gvl_p.etapa_process[0] := 'Secagem';

ELSE
	status:= 20;
END_IF

30:
IF gvl_p.arrStatusEstufas[0].prevFimSeca = systemtime_to_dt(gvl.fbGetLocalSystemTime.systemTime) THEN
	status:= 40;
	
	gvl_p.zona1setpt_019:= gvl_p.arrStatusEstufas[0].tempArm;
	gvl_p.zona2setpt_019:= gvl_p.arrStatusEstufas[0].tempArm;
	
///// GERADOR DE LOG -------------------------------------------------------------
envialog:= 'Armazenagem Iniciada ESTUFA 019';
gvl.logRegister19:= envialog;
	
gvl_p.etapa_process[0] := 'Armazenagem';

ELSE
	status:= 30;
END_IF

40:
IF gvl_p.arrStatusEstufas[0].fimArmazenagem = systemtime_to_dt(gvl.fbGetLocalSystemTime.systemTime) THEN
	status:= 50;
	
	gvl_p.arrStatusEstufas[0].start:= FALSE;
	gvl.bstartchart019:= FALSE;
	gvl.desl_aquecimento_019:= TRUE;
	fbTimeAqueci(in:=TRUE, pt:=T#1S);
	
	gvl_p.etapa_process[0] := '';
	
	gvl_p.arrStatusEstufas[0].statusInicioSecagem := '';
	gvl_p.arrStatusEstufas[0].inicioReator := '';
	gvl_p.arrStatusEstufas[0].statusFimSecagem := '';
	gvl_p.arrStatusEstufas[0].statusFimArmazenagem := '';
	gvl_p.arrStatusEstufas[0].fimSecagem:= DT#1970-1-1-0:0:0;
	gvl.endArm19:= T#0S;
	gvl.endSeca19:= T#0S;
	
	
///// GERADOR DE LOG -------------------------------------------------------------
envialog:= 'Programação Finalizada ESTUFA 019';
gvl.logRegister19:= envialog;

gvl_p.etapa_process[0]:= '';

ELSE
	status:= 40;
END_IF

45:
IF gvl_p.arrStatusEstufas[0].start THEN
status:= 50;
	
	gvl_p.arrStatusEstufas[0].start:= FALSE;
	gvl.bstartchart019:= FALSE;
	gvl.desl_aquecimento_019:= TRUE;
	fbTimeAqueci(in:=TRUE, pt:=T#1S);
	
	gvl_p.etapa_process[0] := '';
	
	gvl_p.arrStatusEstufas[0].statusInicioSecagem := '';
	gvl_p.arrStatusEstufas[0].inicioReator := '';
	gvl_p.arrStatusEstufas[0].statusFimSecagem := '';
	gvl_p.arrStatusEstufas[0].statusFimArmazenagem := '';
	gvl_p.arrStatusEstufas[0].fimSecagem:= DT#1970-1-1-0:0:0;
	gvl.endArm19:= T#0S;
	gvl.endSeca19:= T#0S;
	
///// GERADOR DE LOG -------------------------------------------------------------
envialog:= 'Programação Finalizada ESTUFA 019';
gvl.logRegister19:= envialog;

gvl_p.etapa_process[0]:= '';

ELSE
	status:= 45;
END_IF

50:
IF fbTimeAqueci.Q THEN
	status:= 0;
	
	gvl.desl_aquecimento_019:= FALSE;
	fbTimeAqueci(in:= FALSE);
	
ELSE
	status:= 50;
END_IF
END_CASE

END_PROGRAM

// ---- POUs/Rotina019_Manual.TcPOU
PROGRAM Rotina019_Manual
VAR
	status: INT;
	
	posicaoAtual: STRING;
	envialog: STRING;
	
	fbTimeVentila: ton;
	fbTimeAqueci: ton;
	
	totalManual: STRING(255);
	tempo: STRING(255);
END_VAR

fbTimeVentila();
fbTimeAqueci();

CASE status OF

0:
IF gvl_p.arrStatusEstufas[0].startManual AND STRING_TO_DT(gvl.progInicio[0]) <= systemtime_to_dt(gvl.fbGetLocalSystemTime.systemTime)  THEN
	status:= 5;
	
	gvl.bstartchart019:= TRUE;
	gvl_p.zona1setpt_019:= gvl_p.arr_CustomTime[0,1];
	gvl_p.zona2setpt_019:= gvl_p.arr_CustomTime[0,1];
	gvl.liga_ventilacao_019:= TRUE;
	fbTimeVentila(in:= TRUE, pt:=T#1S);
	
///// GERADOR DE LOG -------------------------------------------------------------

envialog:= 'Programação Manual Iniciada ESTUFA 019';
gvl.logRegister19:= envialog;

	gvl_p.etapa_process[0] := 'Inicializando';
	
ELSE
	status:= 0;
	IF gvl_p.arrStatusEstufas[0].start THEN
		gvl_p.etapa_process[0] := gvl.progInicio[0];
	END_IF
END_IF
5:
IF fbTimeVentila.Q THEN
	status:= 10;
	gvl.liga_ventilacao_019:=FALSE;
	fbTimeVentila(in:= FALSE);
ELSE
	status:= 5;
END_IF

10:
IF gvl.ventilacao_Ligada_019 THEN
	status:= 15;
	
	gvl.liga_aquecimento_019:= TRUE;
	fbTimeAqueci(in:= TRUE, pt:= T#1S);
	
///// GERADOR DE LOG -------------------------------------------------------------

envialog:= 'Aquecendo ESTUFA 019';
gvl.logRegister19:= envialog;
	
	gvl_p.etapa_process[0] := 'Aquecendo';
	
ELSE
	status:= 10;
END_IF

15:
IF fbTimeAqueci.Q THEN
	status:= 20;
	
	gvl.liga_aquecimento_019:= FALSE;
	fbTimeAqueci(in:=false);
ELSE
	status:= 15;
END_IF

20:
IF gvl.zona1atual_019 >= gvl_p.zona1setpt_019 THEN
	status:= 30;
	
gvl.progInicio[0]:= DT_TO_STRING(gvl.somaTempo);
	
///// CALCULAR FIM DA SECAGEM E DA ARMAZENAGEM --------------------------------------------------------------------------------

totalManual:= insert('T#h',INT_TO_STRING(gvl.totalManual[0]),2);
gvl_p.arrStatusEstufas[0].inicioSecagem := STRING_TO_DT(gvl.progInicio[0]);
gvl_p.arrStatusEstufas[0].fimSecagem := STRING_TO_DT(gvl.progInicio[0]) + STRING_TO_TIME(totalManual);
gvl_P.arrStatusEstufas[0].prevFimSeca := gvl_p.arrStatusEstufas[0].fimSecagem;
//gvl_p.arrStatusEstufas[0].fimArmazenagem := gvl_p.arrStatusEstufas[0].fimSecagem + gvl_p.arrStatusEstufas[0].tempoArmazenagem ;

///// IMPRIMIR A HORA E A DATA DO INICIO DA SECAGEM ---------------------------------------------------------------------------
gvl_p.arrStatusEstufas[0].statusInicioSecagem := '';
gvl_p.arrStatusEstufas[0].statusInicioSecagem := concat(gvl_p.arrStatusEstufas[0].statusInicioSecagem,gvl.hora);
gvl_p.arrStatusEstufas[0].statusInicioSecagem := concat(gvl_p.arrStatusEstufas[0].statusInicioSecagem,':');
gvl_p.arrStatusEstufas[0].statusInicioSecagem := concat(gvl_p.arrStatusEstufas[0].statusInicioSecagem,gvl.minuto);
gvl_p.arrStatusEstufas[0].statusInicioSecagem := concat(gvl_p.arrStatusEstufas[0].statusInicioSecagem,' ');
gvl_p.arrStatusEstufas[0].statusInicioSecagem := concat(gvl_p.arrStatusEstufas[0].statusInicioSecagem,gvl.dia);
gvl_p.arrStatusEstufas[0].statusInicioSecagem := concat(gvl_p.arrStatusEstufas[0].statusInicioSecagem,'/');
gvl_p.arrStatusEstufas[0].statusInicioSecagem := concat(gvl_p.arrStatusEstufas[0].statusInicioSecagem,gvl.mes);
gvl_p.arrStatusEstufas[0].statusInicioSecagem := concat(gvl_p.arrStatusEstufas[0].statusInicioSecagem,'/');
gvl_p.arrStatusEstufas[0].statusInicioSecagem := concat(gvl_p.arrStatusEstufas[0].statusInicioSecagem,gvl.ano);

//--------------------REATOR------------------------------------

IF gravarConfigPosicao_Reator.bGravarConfigPosicao_Reator THEN
	gvl_p.arrStatusEstufas[0].inicioReator := '';
	gvl_p.arrStatusEstufas[0].inicioReator := concat(gvl_p.arrStatusEstufas[0].inicioReator,gvl.hora);
	gvl_p.arrStatusEstufas[0].inicioReator := concat(gvl_p.arrStatusEstufas[0].inicioReator,':');
	gvl_p.arrStatusEstufas[0].inicioReator := concat(gvl_p.arrStatusEstufas[0].inicioReator,gvl.minuto);
	gvl_p.arrStatusEstufas[0].inicioReator := concat(gvl_p.arrStatusEstufas[0].inicioReator,' ');
	gvl_p.arrStatusEstufas[0].inicioReator := concat(gvl_p.arrStatusEstufas[0].inicioReator,gvl.dia);
	gvl_p.arrStatusEstufas[0].inicioReator := concat(gvl_p.arrStatusEstufas[0].inicioReator,'/');
	gvl_p.arrStatusEstufas[0].inicioReator := concat(gvl_p.arrStatusEstufas[0].inicioReator,gvl.mes);
	gvl_p.arrStatusEstufas[0].inicioReator := concat(gvl_p.arrStatusEstufas[0].inicioReator,'/');
	gvl_P.arrStatusEstufas[0].inicioReator := concat(gvl_p.arrStatusEstufas[0].inicioReator,gvl.ano);
END_IF

///// DECOMPOR A VARIAVEL FIM DA SECAGEM -----------------------------------------------------------------------------------------------
gvl_p.arrStatusEstufas[0].diaSec := MID(STR:= DT_TO_STRING(gvl_p.arrStatusEstufas[0].fimSecagem) , LEN:= 2, POS:=12);
gvl_p.arrStatusEstufas[0].mesSec := MID(STR:= DT_TO_STRING(gvl_p.arrStatusEstufas[0].fimSecagem), LEN:= 2, POS:=9);
gvl_p.arrStatusEstufas[0].anoSec := MID(STR:= DT_TO_STRING(gvl_p.arrStatusEstufas[0].fimSecagem), LEN:= 2, POS:=6);
gvl_p.arrStatusEstufas[0].horaSec := MID(STR:= DT_TO_STRING(gvl_p.arrStatusEstufas[0].fimSecagem), LEN:= 2, POS:=15);
gvl_p.arrStatusEstufas[0].minutoSec := MID(STR:= DT_TO_STRING(gvl_p.arrStatusEstufas[0].fimSecagem), LEN:= 2, POS:=18);

///// IMPRIMIR A HORA E A DATA DO FIM DA SECAGEM --------------------------------------------------------------------------------------------------------
gvl_p.arrStatusEstufas[0].statusFimSecagem := '';
gvl_p.arrStatusEstufas[0].statusFimSecagem := concat(gvl_p.arrStatusEstufas[0].statusFimSecagem,gvl_p.arrStatusEstufas[0].horaSec);
gvl_p.arrStatusEstufas[0].statusFimSecagem := concat(gvl_p.arrStatusEstufas[0].statusFimSecagem,':');
gvl_p.arrStatusEstufas[0].statusFimSecagem := concat(gvl_p.arrStatusEstufas[0].statusFimSecagem,gvl_p.arrStatusEstufas[0].minutoSec);
gvl_p.arrStatusEstufas[0].statusFimSecagem := concat(gvl_p.arrStatusEstufas[0].statusFimSecagem,' ');
gvl_p.arrStatusEstufas[0].statusFimSecagem := concat(gvl_p.arrStatusEstufas[0].statusFimSecagem,gvl_p.arrStatusEstufas[0].diaSec);
gvl_p.arrStatusEstufas[0].statusFimSecagem := concat(gvl_p.arrStatusEstufas[0].statusFimSecagem,'/');
gvl_p.arrStatusEstufas[0].statusFimSecagem := concat(gvl_p.arrStatusEstufas[0].statusFimSecagem,gvl_p.arrStatusEstufas[0].mesSec);
gvl_p.arrStatusEstufas[0].statusFimSecagem := concat(gvl_p.arrStatusEstufas[0].statusFimSecagem,'/');
gvl_p.arrStatusEstufas[0].statusFimSecagem := concat(gvl_p.arrStatusEstufas[0].statusFimSecagem,gvl_p.arrStatusEstufas[0].anoSec);


///// GERADOR DE LOG -------------------------------------------------------------
envialog:= 'Inicio T1 ESTUFA 019';
gvl.logRegister19:= envialog;

gvl_p.etapa_process[0]:= 'T1';

ELSE
	IF gvl_p.arr_CustomTime[1,1] = 0 THEN
		status:= 45;
	END_IF
	status:= 20;
END_IF

30:
tempo:= insert('T#h',INT_TO_STRING(gvl_p.arr_CustomTime[1,1]),2);
IF STRING_TO_DT(gvl.progInicio[0]) + STRING_TO_TIME(tempo) = systemtime_to_dt(gvl.fbGetLocalSystemTime.systemTime) THEN
	status:= 31;
	
	gvl_p.zona1setpt_019:= gvl_p.arr_CustomTime[0,2];
	gvl_p.zona2setpt_019:= gvl_p.arr_CustomTime[0,2];
	gvl.progInicio[0]:= DT_TO_STRING(STRING_TO_DT(gvl.progInicio[0]) + STRING_TO_TIME(tempo));
	
///// GERADOR DE LOG -------------------------------------------------------------
envialog:= 'Inicio T2 ESTUFA 019';
gvl.logRegister19:= envialog;

gvl_p.etapa_process[0]:= 'T2';
	
ELSE
	status:= 30;
END_IF

31:
tempo:= insert('T#h',INT_TO_STRING(gvl_p.arr_CustomTime[1,2]),2);
IF STRING_TO_DT(gvl.progInicio[0]) + STRING_TO_TIME(tempo) = systemtime_to_dt(gvl.fbGetLocalSystemTime.systemTime) THEN
	status:= 32;
	
	gvl_p.zona1setpt_019:= gvl_p.arr_CustomTime[0,3];
	gvl_p.zona2setpt_019:= gvl_p.arr_CustomTime[0,3];
	gvl.progInicio[0]:= DT_TO_STRING(STRING_TO_DT(gvl.progInicio[0]) + STRING_TO_TIME(tempo));
	
///// GERADOR DE LOG -------------------------------------------------------------
envialog:= 'Inicio T3 ESTUFA 019';
gvl.logRegister19:= envialog;

gvl_p.etapa_process[0]:= 'T3';
	
ELSE
	IF gvl_p.arr_CustomTime[1,2] = 0 THEN
		status:= 45;
	END_IF
	status:= 31;
END_IF

32:
tempo:= insert('T#h',INT_TO_STRING(gvl_p.arr_CustomTime[1,3]),2);
IF STRING_TO_DT(gvl.progInicio[0]) + STRING_TO_TIME(tempo) = systemtime_to_dt(gvl.fbGetLocalSystemTime.systemTime) THEN
	status:= 33;
	
	gvl_p.zona1setpt_019:= gvl_p.arr_CustomTime[0,4];
	gvl_p.zona2setpt_019:= gvl_p.arr_CustomTime[0,4];
	gvl.progInicio[0]:= DT_TO_STRING(STRING_TO_DT(gvl.progInicio[0]) + STRING_TO_TIME(tempo));
	
///// GERADOR DE LOG -------------------------------------------------------------
envialog:= 'Inicio T4 ESTUFA 019';
gvl.logRegister19:= envialog;

gvl_p.etapa_process[0]:= 'T4';
	
ELSE
	IF gvl_p.arr_CustomTime[1,3] = 0 THEN
		status:= 45;
	END_IF
	status:= 32;
END_IF

33:
tempo:= insert('T#h',INT_TO_STRING(gvl_p.arr_CustomTime[1,4]),2);
IF STRING_TO_DT(gvl.progInicio[0]) + STRING_TO_TIME(tempo) = systemtime_to_dt(gvl.fbGetLocalSystemTime.systemTime) THEN
	status:= 34;
	
	gvl_p.zona1setpt_019:= gvl_p.arr_CustomTime[0,5];
	gvl_p.zona2setpt_019:= gvl_p.arr_CustomTime[0,5];
	gvl.progInicio[0]:= DT_TO_STRING(STRING_TO_DT(gvl.progInicio[0]) + STRING_TO_TIME(tempo));
	
///// GERADOR DE LOG -------------------------------------------------------------
envialog:= 'Inicio T5 ESTUFA 019';
gvl.logRegister19:= envialog;

gvl_p.etapa_process[0]:= 'T5';
	
ELSE
	IF gvl_p.arr_CustomTime[1,4] = 0 THEN
		status:= 45;
	END_IF
	status:= 33;
END_IF

34:
tempo:= insert('T#h',INT_TO_STRING(gvl_p.arr_CustomTime[1,5]),2);
IF STRING_TO_DT(gvl.progInicio[0]) + STRING_TO_TIME(tempo) = systemtime_to_dt(gvl.fbGetLocalSystemTime.systemTime) THEN
	status:= 35;
	
	gvl_p.zona1setpt_019:= gvl_p.arr_CustomTime[0,6];
	gvl_p.zona2setpt_019:= gvl_p.arr_CustomTime[0,6];
	gvl.progInicio[0]:= DT_TO_STRING(STRING_TO_DT(gvl.progInicio[0]) + STRING_TO_TIME(tempo));
	
///// GERADOR DE LOG -------------------------------------------------------------
envialog:= 'Inicio T6 ESTUFA 019';
gvl.logRegister19:= envialog;

gvl_p.etapa_process[0]:= 'T6';
	
ELSE
	IF gvl_p.arr_CustomTime[1,5] = 0 THEN
		status:= 45;
	END_IF
	status:= 34;
END_IF

35:
tempo:= insert('T#h',INT_TO_STRING(gvl_p.arr_CustomTime[1,6]),2);
IF STRING_TO_DT(gvl.progInicio[0]) + STRING_TO_TIME(tempo) = systemtime_to_dt(gvl.fbGetLocalSystemTime.systemTime) THEN
	status:= 36;
	
	gvl_p.zona1setpt_019:= gvl_p.arr_CustomTime[0,7];
	gvl_p.zona2setpt_019:= gvl_p.arr_CustomTime[0,7];
	gvl.progInicio[0]:= DT_TO_STRING(STRING_TO_DT(gvl.progInicio[0]) + STRING_TO_TIME(tempo));
	
///// GERADOR DE LOG -------------------------------------------------------------
envialog:= 'Inicio T7 ESTUFA 019';
gvl.logRegister19:= envialog;

gvl_p.etapa_process[0]:= 'T7';
	
ELSE
	IF gvl_p.arr_CustomTime[1,6] = 0 THEN
		status:= 45;
	END_IF
	status:= 35;
END_IF

36:
tempo:= insert('T#h',INT_TO_STRING(gvl_p.arr_CustomTime[1,7]),2);
IF STRING_TO_DT(gvl.progInicio[0]) + STRING_TO_TIME(tempo) = systemtime_to_dt(gvl.fbGetLocalSystemTime.systemTime) THEN
	status:= 37;
	
	gvl_p.zona1setpt_019:= gvl_p.arr_CustomTime[0,8];
	gvl_p.zona2setpt_019:= gvl_p.arr_CustomTime[0,8];
	gvl.progInicio[0]:= DT_TO_STRING(STRING_TO_DT(gvl.progInicio[0]) + STRING_TO_TIME(tempo));
	
///// GERADOR DE LOG -------------------------------------------------------------
envialog:= 'Inicio T8 ESTUFA 019';
gvl.logRegister19:= envialog;

gvl_p.etapa_process[0]:= 'T8';
	
ELSE
	IF gvl_p.arr_CustomTime[1,7] = 0 THEN
		status:= 45;
	END_IF
	status:= 36;
END_IF

37:
tempo:= insert('T#h',INT_TO_STRING(gvl_p.arr_CustomTime[1,8]),2);
IF STRING_TO_DT(gvl.progInicio[0]) + STRING_TO_TIME(tempo) = systemtime_to_dt(gvl.fbGetLocalSystemTime.systemTime) THEN
	status:= 38;
	
	gvl_p.zona1setpt_019:= gvl_p.arr_CustomTime[0,9];
	gvl_p.zona2setpt_019:= gvl_p.arr_CustomTime[0,9];
	gvl.progInicio[0]:= DT_TO_STRING(STRING_TO_DT(gvl.progInicio[0]) + STRING_TO_TIME(tempo));
	
///// GERADOR DE LOG -------------------------------------------------------------
envialog:= 'Inicio T9 ESTUFA 019';
gvl.logRegister19:= envialog;

gvl_p.etapa_process[0]:= 'T9';
	
ELSE
	IF gvl_p.arr_CustomTime[1,8] = 0 THEN
		status:= 45;
	END_IF
	status:= 37;
END_IF

38:
tempo:= insert('T#h',INT_TO_STRING(gvl_p.arr_CustomTime[1,9]),2);
IF STRING_TO_DT(gvl.progInicio[0]) + STRING_TO_TIME(tempo) = systemtime_to_dt(gvl.fbGetLocalSystemTime.systemTime) THEN
	status:= 40;
	
	gvl_p.zona1setpt_019:= gvl_p.arr_CustomTime[0,10];
	gvl_p.zona2setpt_019:= gvl_p.arr_CustomTime[0,10];
	gvl.progInicio[0]:= DT_TO_STRING(STRING_TO_DT(gvl.progInicio[0]) + STRING_TO_TIME(tempo));
	
///// GERADOR DE LOG -------------------------------------------------------------
envialog:= 'Inicio T10 ESTUFA 019';
gvl.logRegister19:= envialog;

gvl_p.etapa_process[0]:= 'T10';
	
ELSE
	IF gvl_p.arr_CustomTime[1,9] = 0 THEN
		status:= 45;
	END_IF
	status:= 38;
END_IF

40:
tempo:= insert('T#h',INT_TO_STRING(gvl_p.arr_CustomTime[1,10]),2);
IF STRING_TO_DT(gvl.progInicio[0]) + STRING_TO_TIME(tempo) = systemtime_to_dt(gvl.fbGetLocalSystemTime.systemTime) THEN
	status:= 50;
	
	gvl_p.arrStatusEstufas[0].startManual:= FALSE;
	gvl.bstartchart019:= FALSE;
	gvl.desl_aquecimento_019:= TRUE;
	fbTimeAqueci(in:=TRUE, pt:=T#1S);
	
	gvl_p.etapa_process[0] := '';
	
	gvl_p.arrStatusEstufas[0].statusInicioSecagem := '';
	gvl_p.arrStatusEstufas[0].inicioReator := '';
	gvl_p.arrStatusEstufas[0].statusFimSecagem := '';
	gvl_p.arrStatusEstufas[0].statusFimArmazenagem := '';
	gvl_p.arrStatusEstufas[0].fimSecagem:= DT#1970-1-1-0:0:0;
	gvl.endArm19:= T#0S;
	gvl.endSeca19:= T#0S;
	
///// GERADOR DE LOG -------------------------------------------------------------
envialog:= 'Programação Finalizada ESTUFA 019';
gvl.logRegister19:= envialog;

gvl_p.etapa_process[0]:= '';

ELSE
	IF gvl_p.arr_CustomTime[1,10] = 0 THEN
		status:= 45;
	END_IF
	status:= 40;
END_IF

45:
IF gvl_p.arrStatusEstufas[0].startManual THEN
status:= 50;
	
	gvl_p.arrStatusEstufas[0].startManual:= FALSE;
	gvl.bstartchart019:= FALSE;
	gvl.desl_aquecimento_019:= TRUE;
	fbTimeAqueci(in:=TRUE, pt:=T#1S);
	
	gvl_p.etapa_process[0] := '';
	
	gvl_p.arrStatusEstufas[0].statusInicioSecagem := '';
	gvl_p.arrStatusEstufas[0].inicioReator := '';
	gvl_p.arrStatusEstufas[0].statusFimSecagem := '';
	gvl_p.arrStatusEstufas[0].statusFimArmazenagem := '';
	gvl_p.arrStatusEstufas[0].fimSecagem:= DT#1970-1-1-0:0:0;
	gvl.endArm19:= T#0S;
	gvl.endSeca19:= T#0S;
	
///// GERADOR DE LOG -------------------------------------------------------------
envialog:= 'Programação Finalizada ESTUFA 019';
gvl.logRegister19:= envialog;

gvl_p.etapa_process[0]:= '';

ELSE
	status:= 45;
END_IF

50:
IF fbTimeAqueci.Q THEN
	status:= 0;
	
	gvl.desl_aquecimento_019:= FALSE;
	fbTimeAqueci(in:= FALSE);
	
ELSE
	status:= 50;
END_IF
END_CASE

END_PROGRAM

// ---- POUs/Rotina020.TcPOU
PROGRAM Rotina020
VAR
	status: INT;
	
	posicaoAtual: STRING;
	envialog: STRING;
	
	fbTimeVentila: ton;
	fbTimeAqueci: ton;
	
	a: INT;
END_VAR

fbTimeVentila();
fbTimeAqueci();
a:=1;

CASE status OF

0:
IF gvl_p.arrStatusEstufas[a].start AND STRING_TO_DT(gvl.progInicio[a]) <= systemtime_to_dt(gvl.fbGetLocalSystemTime.systemTime)  THEN
	status:= 5;
	
	gvl.bstartchart020:= TRUE;
	gvl_p.zona1setpt_020:= gvl_p.arrStatusEstufas[a].tempSeca;
	gvl_p.zona2setpt_020:= gvl_p.arrStatusEstufas[a].tempSeca;
	gvl.liga_ventilacao_020:= TRUE;
	fbTimeVentila(in:= TRUE, pt:=T#1S);

///// GERADOR DE LOG -------------------------------------------------------------

envialog:= 'Inicializando Programação ESTUFA 020';
gvl.logRegister20:= envialog;
	
	gvl_p.etapa_process[a] := 'Inicializando';
	
ELSE
	status:= 0;
	IF gvl_p.arrStatusEstufas[a].start THEN
		gvl_p.etapa_process[a] := gvl.progInicio[a];
	END_IF
END_IF

5:
IF fbTimeVentila.Q THEN
	status:= 10;
	gvl.liga_ventilacao_020:=FALSE;
	fbTimeVentila(in:= FALSE);
ELSE
	status:= 5;
END_IF

10:
IF gvl.ventilacao_Ligada_020 THEN
	status:= 15;
	
	gvl.liga_aquecimento_020:= TRUE;
	fbTimeAqueci(in:= TRUE, pt:= T#1S);
	
///// GERADOR DE LOG -------------------------------------------------------------

envialog:= 'Aquecendo ESTUFA 020';
gvl.logRegister20:= envialog;

	gvl_p.etapa_process[a] := 'Aquecendo';
	
ELSE
	status:= 10;
END_IF

15:
IF fbTimeAqueci.Q THEN
	status:= 20;
	
	gvl.liga_aquecimento_020:= FALSE;
	fbTimeAqueci(in:=false);
ELSE
	status:= 15;
END_IF

20:
IF gvl.zona1atual_020 >= gvl_p.zona1setpt_020 THEN
	status:= 30;

gvl.progInicio[a]:= DT_TO_STRING(gvl.somaTempo);
	
///// CALCULAR FIM DA SECAGEM E DA ARMAZENAGEM --------------------------------------------------------------------------------
gvl_p.arrStatusEstufas[a].inicioSecagem := STRING_TO_DT(gvl.progInicio[a]);
gvl_p.arrStatusEstufas[a].fimSecagem := STRING_TO_DT(gvl.progInicio[a]) + gvl_p.arrStatusEstufas[a].tempoSecagem;
gvl_P.arrStatusEstufas[a].prevFimSeca := gvl_p.arrStatusEstufas[a].fimSecagem;
gvl_p.arrStatusEstufas[a].fimArmazenagem := gvl_p.arrStatusEstufas[a].fimSecagem + gvl_p.arrStatusEstufas[a].tempoArmazenagem ;

///// IMPRIMIR A HORA E A DATA DO INICIO DA SECAGEM ---------------------------------------------------------------------------
gvl_p.arrStatusEstufas[a].statusInicioSecagem := '';
gvl_p.arrStatusEstufas[a].statusInicioSecagem := concat(gvl_p.arrStatusEstufas[a].statusInicioSecagem,gvl.hora);
gvl_p.arrStatusEstufas[a].statusInicioSecagem := concat(gvl_p.arrStatusEstufas[a].statusInicioSecagem,':');
gvl_p.arrStatusEstufas[a].statusInicioSecagem := concat(gvl_p.arrStatusEstufas[a].statusInicioSecagem,gvl.minuto);
gvl_p.arrStatusEstufas[a].statusInicioSecagem := concat(gvl_p.arrStatusEstufas[a].statusInicioSecagem,' ');
gvl_p.arrStatusEstufas[a].statusInicioSecagem := concat(gvl_p.arrStatusEstufas[a].statusInicioSecagem,gvl.dia);
gvl_p.arrStatusEstufas[a].statusInicioSecagem := concat(gvl_p.arrStatusEstufas[a].statusInicioSecagem,'/');
gvl_p.arrStatusEstufas[a].statusInicioSecagem := concat(gvl_p.arrStatusEstufas[a].statusInicioSecagem,gvl.mes);
gvl_p.arrStatusEstufas[a].statusInicioSecagem := concat(gvl_p.arrStatusEstufas[a].statusInicioSecagem,'/');
gvl_p.arrStatusEstufas[a].statusInicioSecagem := concat(gvl_p.arrStatusEstufas[a].statusInicioSecagem,gvl.ano);

//--------------------REATOR------------------------------------

IF gravarConfigPosicao_Reator.bGravarConfigPosicao_Reator THEN
	gvl_p.arrStatusEstufas[a].inicioReator := '';
	gvl_p.arrStatusEstufas[a].inicioReator := concat(gvl_p.arrStatusEstufas[a].inicioReator,gvl.hora);
	gvl_p.arrStatusEstufas[a].inicioReator := concat(gvl_p.arrStatusEstufas[a].inicioReator,':');
	gvl_p.arrStatusEstufas[a].inicioReator := concat(gvl_p.arrStatusEstufas[a].inicioReator,gvl.minuto);
	gvl_p.arrStatusEstufas[a].inicioReator := concat(gvl_p.arrStatusEstufas[a].inicioReator,' ');
	gvl_p.arrStatusEstufas[a].inicioReator := concat(gvl_p.arrStatusEstufas[a].inicioReator,gvl.dia);
	gvl_p.arrStatusEstufas[a].inicioReator := concat(gvl_p.arrStatusEstufas[a].inicioReator,'/');
	gvl_p.arrStatusEstufas[a].inicioReator := concat(gvl_p.arrStatusEstufas[a].inicioReator,gvl.mes);
	gvl_p.arrStatusEstufas[a].inicioReator := concat(gvl_p.arrStatusEstufas[a].inicioReator,'/');
	gvl_P.arrStatusEstufas[a].inicioReator := concat(gvl_p.arrStatusEstufas[a].inicioReator,gvl.ano);
END_IF

///// DECOMPOR A VARIAVEL FIM DA SECAGEM -----------------------------------------------------------------------------------------------
gvl_p.arrStatusEstufas[a].diaSec := MID(STR:= DT_TO_STRING(gvl_p.arrStatusEstufas[a].fimSecagem) , LEN:= 2, POS:=12);
gvl_p.arrStatusEstufas[a].mesSec := MID(STR:= DT_TO_STRING(gvl_p.arrStatusEstufas[a].fimSecagem), LEN:= 2, POS:=9);
gvl_p.arrStatusEstufas[a].anoSec := MID(STR:= DT_TO_STRING(gvl_p.arrStatusEstufas[a].fimSecagem), LEN:= 2, POS:=6);
gvl_p.arrStatusEstufas[a].horaSec := MID(STR:= DT_TO_STRING(gvl_p.arrStatusEstufas[a].fimSecagem), LEN:= 2, POS:=15);
gvl_p.arrStatusEstufas[a].minutoSec := MID(STR:= DT_TO_STRING(gvl_p.arrStatusEstufas[a].fimSecagem), LEN:= 2, POS:=18);

///// IMPRIMIR A HORA E A DATA DO FIM DA SECAGEM --------------------------------------------------------------------------------------------------------
gvl_p.arrStatusEstufas[a].statusFimSecagem := '';
gvl_p.arrStatusEstufas[a].statusFimSecagem := concat(gvl_p.arrStatusEstufas[a].statusFimSecagem,gvl_p.arrStatusEstufas[a].horaSec);
gvl_p.arrStatusEstufas[a].statusFimSecagem := concat(gvl_p.arrStatusEstufas[a].statusFimSecagem,':');
gvl_p.arrStatusEstufas[a].statusFimSecagem := concat(gvl_p.arrStatusEstufas[a].statusFimSecagem,gvl_p.arrStatusEstufas[a].minutoSec);
gvl_p.arrStatusEstufas[a].statusFimSecagem := concat(gvl_p.arrStatusEstufas[a].statusFimSecagem,' ');
gvl_p.arrStatusEstufas[a].statusFimSecagem := concat(gvl_p.arrStatusEstufas[a].statusFimSecagem,gvl_p.arrStatusEstufas[a].diaSec);
gvl_p.arrStatusEstufas[a].statusFimSecagem := concat(gvl_p.arrStatusEstufas[a].statusFimSecagem,'/');
gvl_p.arrStatusEstufas[a].statusFimSecagem := concat(gvl_p.arrStatusEstufas[a].statusFimSecagem,gvl_p.arrStatusEstufas[a].mesSec);
gvl_p.arrStatusEstufas[a].statusFimSecagem := concat(gvl_p.arrStatusEstufas[a].statusFimSecagem,'/');
gvl_p.arrStatusEstufas[a].statusFimSecagem := concat(gvl_p.arrStatusEstufas[a].statusFimSecagem,gvl_p.arrStatusEstufas[a].anoSec);

///// DECOMPOR A VARIAVEL FIM DA ARMAZENAGEM -------------------------------------------------------------------------------------------
gvl_p.arrStatusEstufas[a].diaArm := MID(STR:= DT_TO_STRING(gvl_p.arrStatusEstufas[a].fimArmazenagem) , LEN:= 2, POS:=12);
gvl_p.arrStatusEstufas[a].mesArm := MID(STR:= DT_TO_STRING(gvl_p.arrStatusEstufas[a].fimArmazenagem), LEN:= 2, POS:=9);
gvl_p.arrStatusEstufas[a].anoArm := MID(STR:= DT_TO_STRING(gvl_P.arrStatusEstufas[a].fimArmazenagem), LEN:= 2, POS:=6);
gvl_p.arrStatusEstufas[a].horaArm := MID(STR:= DT_TO_STRING(gvl_P.arrStatusEstufas[a].fimArmazenagem), LEN:= 2, POS:=15);
gvl_p.arrStatusEstufas[a].minutoArm := MID(STR:= DT_TO_STRING(gvl_p.arrStatusEstufas[a].fimArmazenagem), LEN:= 2, POS:=18);

///// IMPRIMIR A HORA E A DATA DO FIM DA ARMAZENAGEM -----------------------------------------------------------------------------------------------------------
gvl_p.arrStatusEstufas[a].statusFimArmazenagem := '';
gvl_p.arrStatusEstufas[a].statusFimArmazenagem := concat(gvl_p.arrStatusEstufas[a].statusFimArmazenagem,gvl_p.arrStatusEstufas[a].horaArm);
gvl_p.arrStatusEstufas[a].statusFimArmazenagem := concat(gvl_p.arrStatusEstufas[a].statusFimArmazenagem,':');
gvl_p.arrStatusEstufas[a].statusFimArmazenagem := concat(gvl_p.arrStatusEstufas[a].statusFimArmazenagem,gvl_p.arrStatusEstufas[a].minutoArm);
gvl_p.arrStatusEstufas[a].statusFimArmazenagem := concat(gvl_p.arrStatusEstufas[a].statusFimArmazenagem,' ');
gvl_p.arrStatusEstufas[a].statusFimArmazenagem := concat(gvl_p.arrStatusEstufas[a].statusFimArmazenagem,gvl_p.arrStatusEstufas[a].diaArm);
gvl_p.arrStatusEstufas[a].statusFimArmazenagem := concat(gvl_p.arrStatusEstufas[a].statusFimArmazenagem,'/');
gvl_p.arrStatusEstufas[a].statusFimArmazenagem := concat(gvl_p.arrStatusEstufas[a].statusFimArmazenagem,gvl_p.arrStatusEstufas[a].mesArm);
gvl_p.arrStatusEstufas[a].statusFimArmazenagem := concat(gvl_p.arrStatusEstufas[a].statusFimArmazenagem,'/');
gvl_p.arrStatusEstufas[a].statusFimArmazenagem := concat(gvl_p.arrStatusEstufas[a].statusFimArmazenagem,gvl_p.arrStatusEstufas[a].anoArm);

///// GERADOR DE LOG -------------------------------------------------------------
envialog:= 'Secagem Iniciada ESTUFA 020';
gvl.logRegister20:= envialog;

gvl_p.etapa_process[a] := 'Secagem';

ELSE
	status:= 20;
END_IF

30:
IF gvl_p.arrStatusEstufas[a].prevFimSeca = systemtime_to_dt(gvl.fbGetLocalSystemTime.systemTime) THEN
	status:= 40;
	
	gvl_p.zona1setpt_020:= gvl_p.arrStatusEstufas[a].tempArm;
	gvl_p.zona2setpt_020:= gvl_p.arrStatusEstufas[a].tempArm;
	
///// GERADOR DE LOG -------------------------------------------------------------
envialog:= 'Armazenagem Iniciada ESTUFA 020';
gvl.logRegister20:= envialog;
	
gvl_p.etapa_process[a] := 'Armazenagem';

ELSE
	status:= 30;
END_IF

40:
IF gvl_p.arrStatusEstufas[a].fimArmazenagem = systemtime_to_dt(gvl.fbGetLocalSystemTime.systemTime) THEN
	status:= 50;
	
	gvl_p.arrStatusEstufas[a].start:= FALSE;
	gvl.bstartchart020:= FALSE;
	gvl.desl_aquecimento_020:= TRUE;
	fbTimeAqueci(in:=TRUE, pt:=T#1S);
	
	gvl_p.etapa_process[a] := '';
	
	gvl_p.arrStatusEstufas[a].statusInicioSecagem := '';
	gvl_p.arrStatusEstufas[a].inicioReator := '';
	gvl_p.arrStatusEstufas[a].statusFimSecagem := '';
	gvl_p.arrStatusEstufas[a].statusFimArmazenagem := '';
	gvl_p.arrStatusEstufas[a].fimSecagem:= DT#1970-1-1-0:0:0;
	gvl.endArm20:= T#0S;
	gvl.endSeca20:= T#0S;
	
	
///// GERADOR DE LOG -------------------------------------------------------------
envialog:= 'Programação Finalizada ESTUFA 020';
gvl.logRegister20:= envialog;

gvl_p.etapa_process[1]:= '';

ELSE
	status:= 40;
END_IF

45:
IF gvl_p.arrStatusEstufas[a].start THEN
status:= 50;
	
	gvl_p.arrStatusEstufas[a].start:= FALSE;
	gvl.bstartchart020:= FALSE;
	gvl.desl_aquecimento_020:= TRUE;
	fbTimeAqueci(in:=TRUE, pt:=T#1S);
	
	gvl_p.etapa_process[a] := '';
	
	gvl_p.arrStatusEstufas[a].statusInicioSecagem := '';
	gvl_p.arrStatusEstufas[a].inicioReator := '';
	gvl_p.arrStatusEstufas[a].statusFimSecagem := '';
	gvl_p.arrStatusEstufas[a].statusFimArmazenagem := '';
	gvl_p.arrStatusEstufas[a].fimSecagem:= DT#1970-1-1-0:0:0;
	gvl.endArm20:= T#0S;
	gvl.endSeca20:= T#0S;
	
///// GERADOR DE LOG -------------------------------------------------------------
envialog:= 'Programação Finalizada ESTUFA 020';
gvl.logRegister20:= envialog;

gvl_p.etapa_process[1]:= '';

ELSE
	status:= 45;
END_IF

50:
IF fbTimeAqueci.Q THEN
	status:= 0;
	
	gvl.desl_aquecimento_020:= FALSE;
	fbTimeAqueci(in:= FALSE);
	
ELSE
	status:= 50;
END_IF
END_CASE

END_PROGRAM

// ---- POUs/Rotina020_Manual.TcPOU
PROGRAM Rotina020_Manual
VAR
	status: INT;
	
	posicaoAtual: STRING;
	envialog: STRING;
	
	fbTimeVentila: ton;
	fbTimeAqueci: ton;
	
	totalManual: STRING(255);
	tempo: STRING(255);
	
	Estufa: INT;
	
END_VAR

fbTimeVentila();
fbTimeAqueci();
Estufa:= 1;

CASE status OF

0:
IF gvl_p.arrStatusEstufas[Estufa].startManual AND STRING_TO_DT(gvl.progInicio[Estufa]) <= systemtime_to_dt(gvl.fbGetLocalSystemTime.systemTime)  THEN
	status:= 5;
	
	gvl.bstartchart020:= TRUE;
	gvl_p.zona1setpt_020:= gvl_p.arr_CustomTime_020[0,1];
	gvl_p.zona2setpt_020:= gvl_p.arr_CustomTime_020[0,1];
	gvl.liga_ventilacao_020:= TRUE;
	fbTimeVentila(in:= TRUE, pt:=T#1S);
	
///// GERADOR DE LOG -------------------------------------------------------------

envialog:= 'Programação Manual Iniciada ESTUFA 020';
gvl.logRegister20:= envialog;

	gvl_p.etapa_process[Estufa] := 'Inicializando';
	
ELSE
	status:= 0;
	IF gvl_p.arrStatusEstufas[Estufa].start THEN
		gvl_p.etapa_process[Estufa] := gvl.progInicio[Estufa];
	END_IF
END_IF
5:
IF fbTimeVentila.Q THEN
	status:= 10;
	gvl.liga_ventilacao_020:=FALSE;
	fbTimeVentila(in:= FALSE);
ELSE
	status:= 5;
END_IF

10:
IF gvl.ventilacao_Ligada_020 THEN
	status:= 15;
	
	gvl.liga_aquecimento_020:= TRUE;
	fbTimeAqueci(in:= TRUE, pt:= T#1S);
	
///// GERADOR DE LOG -------------------------------------------------------------

envialog:= 'Aquecendo ESTUFA 020';
gvl.logRegister20:= envialog;
	gvl_p.etapa_process[Estufa] := 'Aquecendo';
	
ELSE
	status:= 10;
END_IF

15:
IF fbTimeAqueci.Q THEN
	status:= 20;
	
	gvl.liga_aquecimento_020:= FALSE;
	fbTimeAqueci(in:=false);
ELSE
	status:= 15;
END_IF

20:
IF gvl.zona1atual_020 >= gvl_p.zona1setpt_020 THEN
	status:= 30;
	
gvl.progInicio[Estufa]:= DT_TO_STRING(gvl.somaTempo);
	
///// CALCULAR FIM DA SECAGEM E DA ARMAZENAGEM --------------------------------------------------------------------------------

totalManual:= insert('T#h',INT_TO_STRING(gvl.totalManual[Estufa]),2);
gvl_p.arrStatusEstufas[Estufa].inicioSecagem := STRING_TO_DT(gvl.progInicio[Estufa]);
gvl_p.arrStatusEstufas[Estufa].fimSecagem := STRING_TO_DT(gvl.progInicio[Estufa]) + STRING_TO_TIME(totalManual);
gvl_P.arrStatusEstufas[Estufa].prevFimSeca := gvl_p.arrStatusEstufas[Estufa].fimSecagem;
//gvl_p.arrStatusEstufas[0].fimArmazenagem := gvl_p.arrStatusEstufas[0].fimSecagem + gvl_p.arrStatusEstufas[0].tempoArmazenagem ;

///// IMPRIMIR A HORA E A DATA DO INICIO DA SECAGEM ---------------------------------------------------------------------------
gvl_p.arrStatusEstufas[Estufa].statusInicioSecagem := '';
gvl_p.arrStatusEstufas[Estufa].statusInicioSecagem := concat(gvl_p.arrStatusEstufas[Estufa].statusInicioSecagem,gvl.hora);
gvl_p.arrStatusEstufas[Estufa].statusInicioSecagem := concat(gvl_p.arrStatusEstufas[Estufa].statusInicioSecagem,':');
gvl_p.arrStatusEstufas[Estufa].statusInicioSecagem := concat(gvl_p.arrStatusEstufas[Estufa].statusInicioSecagem,gvl.minuto);
gvl_p.arrStatusEstufas[Estufa].statusInicioSecagem := concat(gvl_p.arrStatusEstufas[Estufa].statusInicioSecagem,' ');
gvl_p.arrStatusEstufas[Estufa].statusInicioSecagem := concat(gvl_p.arrStatusEstufas[Estufa].statusInicioSecagem,gvl.dia);
gvl_p.arrStatusEstufas[Estufa].statusInicioSecagem := concat(gvl_p.arrStatusEstufas[Estufa].statusInicioSecagem,'/');
gvl_p.arrStatusEstufas[Estufa].statusInicioSecagem := concat(gvl_p.arrStatusEstufas[Estufa].statusInicioSecagem,gvl.mes);
gvl_p.arrStatusEstufas[Estufa].statusInicioSecagem := concat(gvl_p.arrStatusEstufas[Estufa].statusInicioSecagem,'/');
gvl_p.arrStatusEstufas[Estufa].statusInicioSecagem := concat(gvl_p.arrStatusEstufas[Estufa].statusInicioSecagem,gvl.ano);

//--------------------REATOR------------------------------------

IF gravarConfigPosicao_Reator.bGravarConfigPosicao_Reator THEN
	gvl_p.arrStatusEstufas[Estufa].inicioReator := '';
	gvl_p.arrStatusEstufas[Estufa].inicioReator := concat(gvl_p.arrStatusEstufas[Estufa].inicioReator,gvl.hora);
	gvl_p.arrStatusEstufas[Estufa].inicioReator := concat(gvl_p.arrStatusEstufas[Estufa].inicioReator,':');
	gvl_p.arrStatusEstufas[Estufa].inicioReator := concat(gvl_p.arrStatusEstufas[Estufa].inicioReator,gvl.minuto);
	gvl_p.arrStatusEstufas[Estufa].inicioReator := concat(gvl_p.arrStatusEstufas[Estufa].inicioReator,' ');
	gvl_p.arrStatusEstufas[Estufa].inicioReator := concat(gvl_p.arrStatusEstufas[Estufa].inicioReator,gvl.dia);
	gvl_p.arrStatusEstufas[Estufa].inicioReator := concat(gvl_p.arrStatusEstufas[Estufa].inicioReator,'/');
	gvl_p.arrStatusEstufas[Estufa].inicioReator := concat(gvl_p.arrStatusEstufas[Estufa].inicioReator,gvl.mes);
	gvl_p.arrStatusEstufas[Estufa].inicioReator := concat(gvl_p.arrStatusEstufas[Estufa].inicioReator,'/');
	gvl_P.arrStatusEstufas[Estufa].inicioReator := concat(gvl_p.arrStatusEstufas[Estufa].inicioReator,gvl.ano);
END_IF

///// DECOMPOR A VARIAVEL FIM DA SECAGEM -----------------------------------------------------------------------------------------------
gvl_p.arrStatusEstufas[Estufa].diaSec := MID(STR:= DT_TO_STRING(gvl_p.arrStatusEstufas[Estufa].fimSecagem) , LEN:= 2, POS:=12);
gvl_p.arrStatusEstufas[Estufa].mesSec := MID(STR:= DT_TO_STRING(gvl_p.arrStatusEstufas[Estufa].fimSecagem), LEN:= 2, POS:=9);
gvl_p.arrStatusEstufas[Estufa].anoSec := MID(STR:= DT_TO_STRING(gvl_p.arrStatusEstufas[Estufa].fimSecagem), LEN:= 2, POS:=6);
gvl_p.arrStatusEstufas[Estufa].horaSec := MID(STR:= DT_TO_STRING(gvl_p.arrStatusEstufas[Estufa].fimSecagem), LEN:= 2, POS:=15);
gvl_p.arrStatusEstufas[Estufa].minutoSec := MID(STR:= DT_TO_STRING(gvl_p.arrStatusEstufas[Estufa].fimSecagem), LEN:= 2, POS:=18);

///// IMPRIMIR A HORA E A DATA DO FIM DA SECAGEM --------------------------------------------------------------------------------------------------------
gvl_p.arrStatusEstufas[Estufa].statusFimSecagem := '';
gvl_p.arrStatusEstufas[Estufa].statusFimSecagem := concat(gvl_p.arrStatusEstufas[Estufa].statusFimSecagem,gvl_p.arrStatusEstufas[0].horaSec);
gvl_p.arrStatusEstufas[Estufa].statusFimSecagem := concat(gvl_p.arrStatusEstufas[Estufa].statusFimSecagem,':');
gvl_p.arrStatusEstufas[Estufa].statusFimSecagem := concat(gvl_p.arrStatusEstufas[Estufa].statusFimSecagem,gvl_p.arrStatusEstufas[0].minutoSec);
gvl_p.arrStatusEstufas[Estufa].statusFimSecagem := concat(gvl_p.arrStatusEstufas[Estufa].statusFimSecagem,' ');
gvl_p.arrStatusEstufas[Estufa].statusFimSecagem := concat(gvl_p.arrStatusEstufas[Estufa].statusFimSecagem,gvl_p.arrStatusEstufas[0].diaSec);
gvl_p.arrStatusEstufas[Estufa].statusFimSecagem := concat(gvl_p.arrStatusEstufas[Estufa].statusFimSecagem,'/');
gvl_p.arrStatusEstufas[Estufa].statusFimSecagem := concat(gvl_p.arrStatusEstufas[Estufa].statusFimSecagem,gvl_p.arrStatusEstufas[0].mesSec);
gvl_p.arrStatusEstufas[Estufa].statusFimSecagem := concat(gvl_p.arrStatusEstufas[Estufa].statusFimSecagem,'/');
gvl_p.arrStatusEstufas[Estufa].statusFimSecagem := concat(gvl_p.arrStatusEstufas[Estufa].statusFimSecagem,gvl_p.arrStatusEstufas[0].anoSec);


///// GERADOR DE LOG -------------------------------------------------------------
envialog:= 'Inicio T1 ESTUFA 020';
gvl.logRegister20:= envialog;

gvl_p.etapa_process[1]:= 'T1';

ELSE
	IF gvl_p.arr_CustomTime_020[1,1] = 0 THEN
		status:= 45;
	END_IF
	status:= 20;
END_IF

30:
tempo:= insert('T#h',INT_TO_STRING(gvl_p.arr_CustomTime_020[1,1]),2);
IF STRING_TO_DT(gvl.progInicio[Estufa]) + STRING_TO_TIME(tempo) = systemtime_to_dt(gvl.fbGetLocalSystemTime.systemTime) THEN
	status:= 31;
	
	gvl_p.zona1setpt_020:= gvl_p.arr_CustomTime_020[0,2];
	gvl_p.zona2setpt_020:= gvl_p.arr_CustomTime_020[0,2];
	gvl.progInicio[Estufa]:= DT_TO_STRING(STRING_TO_DT(gvl.progInicio[Estufa]) + STRING_TO_TIME(tempo));
	
///// GERADOR DE LOG -------------------------------------------------------------
envialog:= 'Inicio T2 ESTUFA 020';
gvl.logRegister20:= envialog;

gvl_p.etapa_process[1]:= 'T2';
	
ELSE
	status:= 30;
END_IF

31:
tempo:= insert('T#h',INT_TO_STRING(gvl_p.arr_CustomTime_020[1,2]),2);
IF STRING_TO_DT(gvl.progInicio[Estufa]) + STRING_TO_TIME(tempo) = systemtime_to_dt(gvl.fbGetLocalSystemTime.systemTime) THEN
	status:= 32;
	
	gvl_p.zona1setpt_020:= gvl_p.arr_CustomTime_020[0,3];
	gvl_p.zona2setpt_020:= gvl_p.arr_CustomTime_020[0,3];
	gvl.progInicio[Estufa]:= DT_TO_STRING(STRING_TO_DT(gvl.progInicio[Estufa]) + STRING_TO_TIME(tempo));
	
///// GERADOR DE LOG -------------------------------------------------------------
envialog:= 'Inicio T3 ESTUFA 020';
gvl.logRegister20:= envialog;

gvl_p.etapa_process[1]:= 'T3';
	
ELSE
	IF gvl_p.arr_CustomTime_020[1,2] = 0 THEN
		status:= 45;
	END_IF
	status:= 31;
END_IF

32:
tempo:= insert('T#h',INT_TO_STRING(gvl_p.arr_CustomTime_020[1,3]),2);
IF STRING_TO_DT(gvl.progInicio[Estufa]) + STRING_TO_TIME(tempo) = systemtime_to_dt(gvl.fbGetLocalSystemTime.systemTime) THEN
	status:= 33;
	
	gvl_p.zona1setpt_020:= gvl_p.arr_CustomTime_020[0,4];
	gvl_p.zona2setpt_020:= gvl_p.arr_CustomTime_020[0,4];
	gvl.progInicio[Estufa]:= DT_TO_STRING(STRING_TO_DT(gvl.progInicio[Estufa]) + STRING_TO_TIME(tempo));
	
///// GERADOR DE LOG -------------------------------------------------------------
envialog:= 'Inicio T4 ESTUFA 020';
gvl.logRegister20:= envialog;

gvl_p.etapa_process[1]:= 'T4';
	
ELSE
	IF gvl_p.arr_CustomTime_020[1,3] = 0 THEN
		status:= 45;
	END_IF
	status:= 32;
END_IF

33:
tempo:= insert('T#h',INT_TO_STRING(gvl_p.arr_CustomTime_020[1,4]),2);
IF STRING_TO_DT(gvl.progInicio[Estufa]) + STRING_TO_TIME(tempo) = systemtime_to_dt(gvl.fbGetLocalSystemTime.systemTime) THEN
	status:= 34;
	
	gvl_p.zona1setpt_020:= gvl_p.arr_CustomTime_020[0,5];
	gvl_p.zona2setpt_020:= gvl_p.arr_CustomTime_020[0,5];
	gvl.progInicio[Estufa]:= DT_TO_STRING(STRING_TO_DT(gvl.progInicio[Estufa]) + STRING_TO_TIME(tempo));
	
///// GERADOR DE LOG -------------------------------------------------------------
envialog:= 'Inicio T5 ESTUFA 020';
gvl.logRegister20:= envialog;

gvl_p.etapa_process[1]:= 'T5';
	
ELSE
	IF gvl_p.arr_CustomTime_020[1,4] = 0 THEN
		status:= 45;
	END_IF
	status:= 33;
END_IF

34:
tempo:= insert('T#h',INT_TO_STRING(gvl_p.arr_CustomTime_020[1,5]),2);
IF STRING_TO_DT(gvl.progInicio[Estufa]) + STRING_TO_TIME(tempo) = systemtime_to_dt(gvl.fbGetLocalSystemTime.systemTime) THEN
	status:= 35;
	
	gvl_p.zona1setpt_020:= gvl_p.arr_CustomTime_020[0,6];
	gvl_p.zona2setpt_020:= gvl_p.arr_CustomTime_020[0,6];
	gvl.progInicio[Estufa]:= DT_TO_STRING(STRING_TO_DT(gvl.progInicio[Estufa]) + STRING_TO_TIME(tempo));
	
///// GERADOR DE LOG -------------------------------------------------------------
envialog:= 'Inicio T6 ESTUFA 020';
gvl.logRegister20:= envialog;

gvl_p.etapa_process[1]:= 'T6';
	
ELSE
	IF gvl_p.arr_CustomTime_020[1,5] = 0 THEN
		status:= 45;
	END_IF
	status:= 34;
END_IF

35:
tempo:= insert('T#h',INT_TO_STRING(gvl_p.arr_CustomTime_020[1,6]),2);
IF STRING_TO_DT(gvl.progInicio[Estufa]) + STRING_TO_TIME(tempo) = systemtime_to_dt(gvl.fbGetLocalSystemTime.systemTime) THEN
	status:= 36;
	
	gvl_p.zona1setpt_020:= gvl_p.arr_CustomTime_020[0,7];
	gvl_p.zona2setpt_020:= gvl_p.arr_CustomTime_020[0,7];
	gvl.progInicio[Estufa]:= DT_TO_STRING(STRING_TO_DT(gvl.progInicio[Estufa]) + STRING_TO_TIME(tempo));
	
///// GERADOR DE LOG -------------------------------------------------------------
envialog:= 'Inicio T7 ESTUFA 020';
gvl.logRegister20:= envialog;

gvl_p.etapa_process[1]:= 'T7';
	
ELSE
	IF gvl_p.arr_CustomTime_020[1,6] = 0 THEN
		status:= 45;
	END_IF
	status:= 35;
END_IF

36:
tempo:= insert('T#h',INT_TO_STRING(gvl_p.arr_CustomTime_020[1,7]),2);
IF STRING_TO_DT(gvl.progInicio[Estufa]) + STRING_TO_TIME(tempo) = systemtime_to_dt(gvl.fbGetLocalSystemTime.systemTime) THEN
	status:= 37;
	
	gvl_p.zona1setpt_020:= gvl_p.arr_CustomTime_020[0,8];
	gvl_p.zona2setpt_020:= gvl_p.arr_CustomTime_020[0,8];
	gvl.progInicio[Estufa]:= DT_TO_STRING(STRING_TO_DT(gvl.progInicio[Estufa]) + STRING_TO_TIME(tempo));
	
///// GERADOR DE LOG -------------------------------------------------------------
envialog:= 'Inicio T8 ESTUFA 020';
gvl.logRegister20:= envialog;

gvl_p.etapa_process[1]:= 'T8';
	
ELSE
	IF gvl_p.arr_CustomTime_020[1,7] = 0 THEN
		status:= 45;
	END_IF
	status:= 36;
END_IF

37:
tempo:= insert('T#h',INT_TO_STRING(gvl_p.arr_CustomTime_020[1,8]),2);
IF STRING_TO_DT(gvl.progInicio[Estufa]) + STRING_TO_TIME(tempo) = systemtime_to_dt(gvl.fbGetLocalSystemTime.systemTime) THEN
	status:= 38;
	
	gvl_p.zona1setpt_020:= gvl_p.arr_CustomTime_020[0,9];
	gvl_p.zona2setpt_020:= gvl_p.arr_CustomTime_020[0,9];
	gvl.progInicio[Estufa]:= DT_TO_STRING(STRING_TO_DT(gvl.progInicio[Estufa]) + STRING_TO_TIME(tempo));
	
///// GERADOR DE LOG -------------------------------------------------------------
envialog:= 'Inicio T9 ESTUFA 020';
gvl.logRegister20:= envialog;

gvl_p.etapa_process[1]:= 'T9';
	
ELSE
	IF gvl_p.arr_CustomTime_020[1,8] = 0 THEN
		status:= 45;
	END_IF
	status:= 37;
END_IF

38:
tempo:= insert('T#h',INT_TO_STRING(gvl_p.arr_CustomTime_020[1,9]),2);
IF STRING_TO_DT(gvl.progInicio[Estufa]) + STRING_TO_TIME(tempo) = systemtime_to_dt(gvl.fbGetLocalSystemTime.systemTime) THEN
	status:= 40;
	
	gvl_p.zona1setpt_020:= gvl_p.arr_CustomTime_020[0,10];
	gvl_p.zona2setpt_020:= gvl_p.arr_CustomTime_020[0,10];
	gvl.progInicio[Estufa]:= DT_TO_STRING(STRING_TO_DT(gvl.progInicio[Estufa]) + STRING_TO_TIME(tempo));
	
///// GERADOR DE LOG -------------------------------------------------------------
envialog:= 'Inicio T10 ESTUFA 020';
gvl.logRegister20:= envialog;

gvl_p.etapa_process[1]:= 'T10';
	
ELSE
	IF gvl_p.arr_CustomTime_020[1,9] = 0 THEN
		status:= 45;
	END_IF
	status:= 38;
END_IF

40:
tempo:= insert('T#h',INT_TO_STRING(gvl_p.arr_CustomTime_020[1,10]),2);
IF STRING_TO_DT(gvl.progInicio[Estufa]) + STRING_TO_TIME(tempo) = systemtime_to_dt(gvl.fbGetLocalSystemTime.systemTime) THEN
	status:= 50;
	
	gvl_p.arrStatusEstufas[Estufa].startManual:= FALSE;
	gvl.bstartchart020:= FALSE;
	gvl.desl_aquecimento_020:= TRUE;
	fbTimeAqueci(in:=TRUE, pt:=T#1S);
	
	gvl_p.etapa_process[Estufa] := '';
	
	gvl_p.arrStatusEstufas[Estufa].statusInicioSecagem := '';
	gvl_p.arrStatusEstufas[Estufa].inicioReator := '';
	gvl_p.arrStatusEstufas[Estufa].statusFimSecagem := '';
	gvl_p.arrStatusEstufas[Estufa].statusFimArmazenagem := '';
	gvl_p.arrStatusEstufas[Estufa].fimSecagem:= DT#1970-1-1-0:0:0;
	gvl.endArm20:= T#0S;
	gvl.endSeca20:= T#0S;
	
///// GERADOR DE LOG -------------------------------------------------------------
envialog:= 'Programação Finalizada ESTUFA 020';
gvl.logRegister20:= envialog;

gvl_p.etapa_process[1]:= '';

ELSE
	IF gvl_p.arr_CustomTime_020[1,10] = 0 THEN
		status:= 45;
	END_IF
	status:= 40;
END_IF

45:
IF gvl_p.arrStatusEstufas[Estufa].startManual THEN
status:= 50;
	
	gvl_p.arrStatusEstufas[Estufa].startManual:= FALSE;
	gvl.bstartchart020:= FALSE;
	gvl.desl_aquecimento_020:= TRUE;
	fbTimeAqueci(in:=TRUE, pt:=T#1S);
	
	gvl_p.etapa_process[Estufa] := '';
	
	gvl_p.arrStatusEstufas[Estufa].statusInicioSecagem := '';
	gvl_p.arrStatusEstufas[Estufa].inicioReator := '';
	gvl_p.arrStatusEstufas[Estufa].statusFimSecagem := '';
	gvl_p.arrStatusEstufas[Estufa].statusFimArmazenagem := '';
	gvl_p.arrStatusEstufas[Estufa].fimSecagem:= DT#1970-1-1-0:0:0;
	gvl.endArm20:= T#0S;
	gvl.endSeca20:= T#0S;
	
///// GERADOR DE LOG -------------------------------------------------------------
envialog:= 'Programação Finalizada ESTUFA 020';
gvl.logRegister20:= envialog;

gvl_p.etapa_process[1]:= '';

ELSE
	status:= 45;
END_IF

50:
IF fbTimeAqueci.Q THEN
	status:= 0;
	
	gvl.desl_aquecimento_020:= FALSE;
	fbTimeAqueci(in:= FALSE);
	
ELSE
	status:= 50;
END_IF
END_CASE

END_PROGRAM

// ---- POUs/Rotina021.TcPOU
PROGRAM Rotina021
VAR
	status: INT;
	
	posicaoAtual: STRING;
	envialog: STRING;
	
	fbTimeVentila: ton;
	fbTimeAqueci: ton;
	
	a: INT;
END_VAR

fbTimeVentila();
fbTimeAqueci();
a:=2;

CASE status OF

0:
IF gvl_p.arrStatusEstufas[a].start AND STRING_TO_DT(gvl.progInicio[a]) <= systemtime_to_dt(gvl.fbGetLocalSystemTime.systemTime)  THEN
	status:= 5;
	
	gvl.bstartchart021:= TRUE;
	gvl_p.zona1setpt_021:= gvl_p.arrStatusEstufas[a].tempSeca;
	gvl_p.zona2setpt_021:= gvl_p.arrStatusEstufas[a].tempSeca;
	gvl.liga_ventilacao_021:= TRUE;
	fbTimeVentila(in:= TRUE, pt:=T#1S);
	
	
///// GERADOR DE LOG -------------------------------------------------------------

envialog:= 'Inicializando Programação ESTUFA 021';
gvl.logRegister21:= envialog;

	gvl_p.etapa_process[a] := 'Inicializando';
	
ELSE
	status:= 0;
	IF gvl_p.arrStatusEstufas[a].start THEN
		gvl_p.etapa_process[a] := gvl.progInicio[a];
	END_IF
END_IF
5:
IF fbTimeVentila.Q THEN
	status:= 10;
	gvl.liga_ventilacao_021:=FALSE;
	fbTimeVentila(in:= FALSE);
ELSE
	status:= 5;
END_IF

10:
IF gvl.ventilacao_Ligada_021 THEN
	status:= 15;
	
	gvl.liga_aquecimento_021:= TRUE;
	fbTimeAqueci(in:= TRUE, pt:= T#1S);
	
///// GERADOR DE LOG -------------------------------------------------------------

envialog:= 'Aquecendo ESTUFA 021';
gvl.logRegister21:= envialog;

	gvl_p.etapa_process[a] := 'Aquecendo';
	
ELSE
	status:= 10;
END_IF

15:
IF fbTimeAqueci.Q THEN
	status:= 20;
	
	gvl.liga_aquecimento_021:= FALSE;
	fbTimeAqueci(in:=false);
ELSE
	status:= 15;
END_IF

20:
IF gvl.zona1atual_021 >= gvl_p.zona1setpt_021 THEN
	status:= 30;
	
gvl.progInicio[a]:= DT_TO_STRING(gvl.somaTempo);	
	
///// CALCULAR FIM DA SECAGEM E DA ARMAZENAGEM --------------------------------------------------------------------------------
gvl_p.arrStatusEstufas[a].inicioSecagem := STRING_TO_DT(gvl.progInicio[a]);
gvl_p.arrStatusEstufas[a].fimSecagem := STRING_TO_DT(gvl.progInicio[a]) + gvl_p.arrStatusEstufas[a].tempoSecagem;
gvl_P.arrStatusEstufas[a].prevFimSeca := gvl_p.arrStatusEstufas[a].fimSecagem;
gvl_p.arrStatusEstufas[a].fimArmazenagem := gvl_p.arrStatusEstufas[a].fimSecagem + gvl_p.arrStatusEstufas[a].tempoArmazenagem ;

///// IMPRIMIR A HORA E A DATA DO INICIO DA SECAGEM ---------------------------------------------------------------------------
gvl_p.arrStatusEstufas[a].statusInicioSecagem := '';
gvl_p.arrStatusEstufas[a].statusInicioSecagem := concat(gvl_p.arrStatusEstufas[a].statusInicioSecagem,gvl.hora);
gvl_p.arrStatusEstufas[a].statusInicioSecagem := concat(gvl_p.arrStatusEstufas[a].statusInicioSecagem,':');
gvl_p.arrStatusEstufas[a].statusInicioSecagem := concat(gvl_p.arrStatusEstufas[a].statusInicioSecagem,gvl.minuto);
gvl_p.arrStatusEstufas[a].statusInicioSecagem := concat(gvl_p.arrStatusEstufas[a].statusInicioSecagem,' ');
gvl_p.arrStatusEstufas[a].statusInicioSecagem := concat(gvl_p.arrStatusEstufas[a].statusInicioSecagem,gvl.dia);
gvl_p.arrStatusEstufas[a].statusInicioSecagem := concat(gvl_p.arrStatusEstufas[a].statusInicioSecagem,'/');
gvl_p.arrStatusEstufas[a].statusInicioSecagem := concat(gvl_p.arrStatusEstufas[a].statusInicioSecagem,gvl.mes);
gvl_p.arrStatusEstufas[a].statusInicioSecagem := concat(gvl_p.arrStatusEstufas[a].statusInicioSecagem,'/');
gvl_p.arrStatusEstufas[a].statusInicioSecagem := concat(gvl_p.arrStatusEstufas[a].statusInicioSecagem,gvl.ano);

//--------------------REATOR------------------------------------

IF gravarConfigPosicao_Reator.bGravarConfigPosicao_Reator THEN
	gvl_p.arrStatusEstufas[a].inicioReator := '';
	gvl_p.arrStatusEstufas[a].inicioReator := concat(gvl_p.arrStatusEstufas[a].inicioReator,gvl.hora);
	gvl_p.arrStatusEstufas[a].inicioReator := concat(gvl_p.arrStatusEstufas[a].inicioReator,':');
	gvl_p.arrStatusEstufas[a].inicioReator := concat(gvl_p.arrStatusEstufas[a].inicioReator,gvl.minuto);
	gvl_p.arrStatusEstufas[a].inicioReator := concat(gvl_p.arrStatusEstufas[a].inicioReator,' ');
	gvl_p.arrStatusEstufas[a].inicioReator := concat(gvl_p.arrStatusEstufas[a].inicioReator,gvl.dia);
	gvl_p.arrStatusEstufas[a].inicioReator := concat(gvl_p.arrStatusEstufas[a].inicioReator,'/');
	gvl_p.arrStatusEstufas[a].inicioReator := concat(gvl_p.arrStatusEstufas[a].inicioReator,gvl.mes);
	gvl_p.arrStatusEstufas[a].inicioReator := concat(gvl_p.arrStatusEstufas[a].inicioReator,'/');
	gvl_P.arrStatusEstufas[a].inicioReator := concat(gvl_p.arrStatusEstufas[a].inicioReator,gvl.ano);
END_IF

///// DECOMPOR A VARIAVEL FIM DA SECAGEM -----------------------------------------------------------------------------------------------
gvl_p.arrStatusEstufas[a].diaSec := MID(STR:= DT_TO_STRING(gvl_p.arrStatusEstufas[a].fimSecagem) , LEN:= 2, POS:=12);
gvl_p.arrStatusEstufas[a].mesSec := MID(STR:= DT_TO_STRING(gvl_p.arrStatusEstufas[a].fimSecagem), LEN:= 2, POS:=9);
gvl_p.arrStatusEstufas[a].anoSec := MID(STR:= DT_TO_STRING(gvl_p.arrStatusEstufas[a].fimSecagem), LEN:= 2, POS:=6);
gvl_p.arrStatusEstufas[a].horaSec := MID(STR:= DT_TO_STRING(gvl_p.arrStatusEstufas[a].fimSecagem), LEN:= 2, POS:=15);
gvl_p.arrStatusEstufas[a].minutoSec := MID(STR:= DT_TO_STRING(gvl_p.arrStatusEstufas[a].fimSecagem), LEN:= 2, POS:=18);

///// IMPRIMIR A HORA E A DATA DO FIM DA SECAGEM --------------------------------------------------------------------------------------------------------
gvl_p.arrStatusEstufas[a].statusFimSecagem := '';
gvl_p.arrStatusEstufas[a].statusFimSecagem := concat(gvl_p.arrStatusEstufas[a].statusFimSecagem,gvl_p.arrStatusEstufas[a].horaSec);
gvl_p.arrStatusEstufas[a].statusFimSecagem := concat(gvl_p.arrStatusEstufas[a].statusFimSecagem,':');
gvl_p.arrStatusEstufas[a].statusFimSecagem := concat(gvl_p.arrStatusEstufas[a].statusFimSecagem,gvl_p.arrStatusEstufas[a].minutoSec);
gvl_p.arrStatusEstufas[a].statusFimSecagem := concat(gvl_p.arrStatusEstufas[a].statusFimSecagem,' ');
gvl_p.arrStatusEstufas[a].statusFimSecagem := concat(gvl_p.arrStatusEstufas[a].statusFimSecagem,gvl_p.arrStatusEstufas[a].diaSec);
gvl_p.arrStatusEstufas[a].statusFimSecagem := concat(gvl_p.arrStatusEstufas[a].statusFimSecagem,'/');
gvl_p.arrStatusEstufas[a].statusFimSecagem := concat(gvl_p.arrStatusEstufas[a].statusFimSecagem,gvl_p.arrStatusEstufas[a].mesSec);
gvl_p.arrStatusEstufas[a].statusFimSecagem := concat(gvl_p.arrStatusEstufas[a].statusFimSecagem,'/');
gvl_p.arrStatusEstufas[a].statusFimSecagem := concat(gvl_p.arrStatusEstufas[a].statusFimSecagem,gvl_p.arrStatusEstufas[a].anoSec);

///// DECOMPOR A VARIAVEL FIM DA ARMAZENAGEM -------------------------------------------------------------------------------------------
gvl_p.arrStatusEstufas[a].diaArm := MID(STR:= DT_TO_STRING(gvl_p.arrStatusEstufas[a].fimArmazenagem) , LEN:= 2, POS:=12);
gvl_p.arrStatusEstufas[a].mesArm := MID(STR:= DT_TO_STRING(gvl_p.arrStatusEstufas[a].fimArmazenagem), LEN:= 2, POS:=9);
gvl_p.arrStatusEstufas[a].anoArm := MID(STR:= DT_TO_STRING(gvl_P.arrStatusEstufas[a].fimArmazenagem), LEN:= 2, POS:=6);
gvl_p.arrStatusEstufas[a].horaArm := MID(STR:= DT_TO_STRING(gvl_P.arrStatusEstufas[a].fimArmazenagem), LEN:= 2, POS:=15);
gvl_p.arrStatusEstufas[a].minutoArm := MID(STR:= DT_TO_STRING(gvl_p.arrStatusEstufas[a].fimArmazenagem), LEN:= 2, POS:=18);

///// IMPRIMIR A HORA E A DATA DO FIM DA ARMAZENAGEM -----------------------------------------------------------------------------------------------------------
gvl_p.arrStatusEstufas[a].statusFimArmazenagem := '';
gvl_p.arrStatusEstufas[a].statusFimArmazenagem := concat(gvl_p.arrStatusEstufas[a].statusFimArmazenagem,gvl_p.arrStatusEstufas[a].horaArm);
gvl_p.arrStatusEstufas[a].statusFimArmazenagem := concat(gvl_p.arrStatusEstufas[a].statusFimArmazenagem,':');
gvl_p.arrStatusEstufas[a].statusFimArmazenagem := concat(gvl_p.arrStatusEstufas[a].statusFimArmazenagem,gvl_p.arrStatusEstufas[a].minutoArm);
gvl_p.arrStatusEstufas[a].statusFimArmazenagem := concat(gvl_p.arrStatusEstufas[a].statusFimArmazenagem,' ');
gvl_p.arrStatusEstufas[a].statusFimArmazenagem := concat(gvl_p.arrStatusEstufas[a].statusFimArmazenagem,gvl_p.arrStatusEstufas[a].diaArm);
gvl_p.arrStatusEstufas[a].statusFimArmazenagem := concat(gvl_p.arrStatusEstufas[a].statusFimArmazenagem,'/');
gvl_p.arrStatusEstufas[a].statusFimArmazenagem := concat(gvl_p.arrStatusEstufas[a].statusFimArmazenagem,gvl_p.arrStatusEstufas[a].mesArm);
gvl_p.arrStatusEstufas[a].statusFimArmazenagem := concat(gvl_p.arrStatusEstufas[a].statusFimArmazenagem,'/');
gvl_p.arrStatusEstufas[a].statusFimArmazenagem := concat(gvl_p.arrStatusEstufas[a].statusFimArmazenagem,gvl_p.arrStatusEstufas[a].anoArm);

///// GERADOR DE LOG -------------------------------------------------------------
envialog:= 'Secagem Iniciada ESTUFA 021';
gvl.logRegister21:= envialog;

gvl_p.etapa_process[a] := 'Secagem';

ELSE
	status:= 20;
END_IF

30:
IF gvl_p.arrStatusEstufas[a].prevFimSeca = systemtime_to_dt(gvl.fbGetLocalSystemTime.systemTime) THEN
	status:= 40;
	
	gvl_p.zona1setpt_021:= gvl_p.arrStatusEstufas[a].tempArm;
	gvl_p.zona2setpt_021:= gvl_p.arrStatusEstufas[a].tempArm;
	
///// GERADOR DE LOG -------------------------------------------------------------
envialog:= 'Armazenagem Iniciada ESTUFA 021';
gvl.logRegister21:= envialog;

	
gvl_p.etapa_process[a] := 'Armazenagem';

ELSE
	status:= 30;
END_IF

40:
IF gvl_p.arrStatusEstufas[a].fimArmazenagem = systemtime_to_dt(gvl.fbGetLocalSystemTime.systemTime) THEN
	status:= 50;
	
	gvl_p.arrStatusEstufas[a].start:= FALSE;
	gvl.bstartchart021:= FALSE;
	gvl.desl_aquecimento_021:= TRUE;
	fbTimeAqueci(in:=TRUE, pt:=T#1S);
	
	gvl_p.etapa_process[a] := '';
	
	gvl_p.arrStatusEstufas[a].statusInicioSecagem := '';
	gvl_p.arrStatusEstufas[a].inicioReator := '';
	gvl_p.arrStatusEstufas[a].statusFimSecagem := '';
	gvl_p.arrStatusEstufas[a].statusFimArmazenagem := '';
	gvl_p.arrStatusEstufas[a].fimSecagem:= DT#1970-1-1-0:0:0;
	gvl.endArm21:= T#0S;
	gvl.endSeca21:= T#0S;
	
///// GERADOR DE LOG -------------------------------------------------------------
envialog:= 'Programação Finalizada ESTUFA 021';
gvl.logRegister21:= envialog;

gvl_p.etapa_process[2]:= '';

ELSE
	status:= 40;
END_IF

45:
IF gvl_p.arrStatusEstufas[a].start THEN
status:= 50;
	
	gvl_p.arrStatusEstufas[a].start:= FALSE;
	gvl.bstartchart021:= FALSE;
	gvl.desl_aquecimento_021:= TRUE;
	fbTimeAqueci(in:=TRUE, pt:=T#1S);
	
	gvl_p.etapa_process[a] := '';
	
	gvl_p.arrStatusEstufas[a].statusInicioSecagem := '';
	gvl_p.arrStatusEstufas[a].inicioReator := '';
	gvl_p.arrStatusEstufas[a].statusFimSecagem := '';
	gvl_p.arrStatusEstufas[a].statusFimArmazenagem := '';
	gvl_p.arrStatusEstufas[a].fimSecagem:= DT#1970-1-1-0:0:0;
	gvl.endArm21:= T#0S;
	gvl.endSeca21:= T#0S;
	
///// GERADOR DE LOG -------------------------------------------------------------
envialog:= 'Programação Finalizada ESTUFA 021';
gvl.logRegister21:= envialog;

gvl_p.etapa_process[2]:= '';

ELSE
	status:= 45;
END_IF

50:
IF fbTimeAqueci.Q THEN
	status:= 0;
	
	gvl.desl_aquecimento_021:= FALSE;
	fbTimeAqueci(in:= FALSE);
	
ELSE
	status:= 50;
END_IF
END_CASE

END_PROGRAM

// ---- POUs/Rotina021_Manual.TcPOU
PROGRAM Rotina021_Manual
VAR
	status: INT;
	
	posicaoAtual: STRING;
	envialog: STRING;
	
	fbTimeVentila: ton;
	fbTimeAqueci: ton;
	
	totalManual: STRING(255);
	tempo: STRING(255);
	
	Estufa: INT;
	
END_VAR

fbTimeVentila();
fbTimeAqueci();
Estufa:= 2;

CASE status OF

0:
IF gvl_p.arrStatusEstufas[Estufa].startManual AND STRING_TO_DT(gvl.progInicio[Estufa]) <= systemtime_to_dt(gvl.fbGetLocalSystemTime.systemTime)  THEN
	status:= 5;
	
	gvl.bstartchart021:= TRUE;
	gvl_p.zona1setpt_021:= gvl_p.arr_CustomTime_021[0,1];
	gvl_p.zona2setpt_021:= gvl_p.arr_CustomTime_021[0,1];
	gvl.liga_ventilacao_021:= TRUE;
	fbTimeVentila(in:= TRUE, pt:=T#1S);
	
///// GERADOR DE LOG -------------------------------------------------------------

envialog:= 'Programação Manual Iniciada ESTUFA 021';
gvl.logRegister21:= envialog;
	
	gvl_p.etapa_process[Estufa] := 'Inicializando';
	
ELSE
	status:= 0;
	IF gvl_p.arrStatusEstufas[Estufa].start THEN
		gvl_p.etapa_process[Estufa] := gvl.progInicio[Estufa];
	END_IF
END_IF
5:
IF fbTimeVentila.Q THEN
	status:= 10;
	gvl.liga_ventilacao_021:=FALSE;
	fbTimeVentila(in:= FALSE);
ELSE
	status:= 5;
END_IF

10:
IF gvl.ventilacao_Ligada_021 THEN
	status:= 15;
	
	gvl.liga_aquecimento_021:= TRUE;
	fbTimeAqueci(in:= TRUE, pt:= T#1S);
	
///// GERADOR DE LOG -------------------------------------------------------------

envialog:= 'Aquecendo ESTUFA 021';
gvl.logRegister21:= envialog;

	gvl_p.etapa_process[Estufa] := 'Aquecendo';
	
ELSE
	status:= 10;
END_IF

15:
IF fbTimeAqueci.Q THEN
	status:= 20;
	
	gvl.liga_aquecimento_021:= FALSE;
	fbTimeAqueci(in:=false);
ELSE
	status:= 15;
END_IF

20:
IF gvl.zona1atual_021 >= gvl_p.zona1setpt_021 THEN
	status:= 30;
	
gvl.progInicio[Estufa]:= DT_TO_STRING(gvl.somaTempo);
	
///// CALCULAR FIM DA SECAGEM E DA ARMAZENAGEM --------------------------------------------------------------------------------

totalManual:= insert('T#h',INT_TO_STRING(gvl.totalManual[Estufa]),2);
gvl_p.arrStatusEstufas[Estufa].inicioSecagem := STRING_TO_DT(gvl.progInicio[Estufa]);
gvl_p.arrStatusEstufas[Estufa].fimSecagem := STRING_TO_DT(gvl.progInicio[Estufa]) + STRING_TO_TIME(totalManual);
gvl_P.arrStatusEstufas[Estufa].prevFimSeca := gvl_p.arrStatusEstufas[Estufa].fimSecagem;
//gvl_p.arrStatusEstufas[0].fimArmazenagem := gvl_p.arrStatusEstufas[0].fimSecagem + gvl_p.arrStatusEstufas[0].tempoArmazenagem ;

///// IMPRIMIR A HORA E A DATA DO INICIO DA SECAGEM ---------------------------------------------------------------------------
gvl_p.arrStatusEstufas[Estufa].statusInicioSecagem := '';
gvl_p.arrStatusEstufas[Estufa].statusInicioSecagem := concat(gvl_p.arrStatusEstufas[Estufa].statusInicioSecagem,gvl.hora);
gvl_p.arrStatusEstufas[Estufa].statusInicioSecagem := concat(gvl_p.arrStatusEstufas[Estufa].statusInicioSecagem,':');
gvl_p.arrStatusEstufas[Estufa].statusInicioSecagem := concat(gvl_p.arrStatusEstufas[Estufa].statusInicioSecagem,gvl.minuto);
gvl_p.arrStatusEstufas[Estufa].statusInicioSecagem := concat(gvl_p.arrStatusEstufas[Estufa].statusInicioSecagem,' ');
gvl_p.arrStatusEstufas[Estufa].statusInicioSecagem := concat(gvl_p.arrStatusEstufas[Estufa].statusInicioSecagem,gvl.dia);
gvl_p.arrStatusEstufas[Estufa].statusInicioSecagem := concat(gvl_p.arrStatusEstufas[Estufa].statusInicioSecagem,'/');
gvl_p.arrStatusEstufas[Estufa].statusInicioSecagem := concat(gvl_p.arrStatusEstufas[Estufa].statusInicioSecagem,gvl.mes);
gvl_p.arrStatusEstufas[Estufa].statusInicioSecagem := concat(gvl_p.arrStatusEstufas[Estufa].statusInicioSecagem,'/');
gvl_p.arrStatusEstufas[Estufa].statusInicioSecagem := concat(gvl_p.arrStatusEstufas[Estufa].statusInicioSecagem,gvl.ano);

//--------------------REATOR------------------------------------

IF gravarConfigPosicao_Reator.bGravarConfigPosicao_Reator THEN
	gvl_p.arrStatusEstufas[Estufa].inicioReator := '';
	gvl_p.arrStatusEstufas[Estufa].inicioReator := concat(gvl_p.arrStatusEstufas[Estufa].inicioReator,gvl.hora);
	gvl_p.arrStatusEstufas[Estufa].inicioReator := concat(gvl_p.arrStatusEstufas[Estufa].inicioReator,':');
	gvl_p.arrStatusEstufas[Estufa].inicioReator := concat(gvl_p.arrStatusEstufas[Estufa].inicioReator,gvl.minuto);
	gvl_p.arrStatusEstufas[Estufa].inicioReator := concat(gvl_p.arrStatusEstufas[Estufa].inicioReator,' ');
	gvl_p.arrStatusEstufas[Estufa].inicioReator := concat(gvl_p.arrStatusEstufas[Estufa].inicioReator,gvl.dia);
	gvl_p.arrStatusEstufas[Estufa].inicioReator := concat(gvl_p.arrStatusEstufas[Estufa].inicioReator,'/');
	gvl_p.arrStatusEstufas[Estufa].inicioReator := concat(gvl_p.arrStatusEstufas[Estufa].inicioReator,gvl.mes);
	gvl_p.arrStatusEstufas[Estufa].inicioReator := concat(gvl_p.arrStatusEstufas[Estufa].inicioReator,'/');
	gvl_P.arrStatusEstufas[Estufa].inicioReator := concat(gvl_p.arrStatusEstufas[Estufa].inicioReator,gvl.ano);
END_IF

///// DECOMPOR A VARIAVEL FIM DA SECAGEM -----------------------------------------------------------------------------------------------
gvl_p.arrStatusEstufas[Estufa].diaSec := MID(STR:= DT_TO_STRING(gvl_p.arrStatusEstufas[Estufa].fimSecagem) , LEN:= 2, POS:=12);
gvl_p.arrStatusEstufas[Estufa].mesSec := MID(STR:= DT_TO_STRING(gvl_p.arrStatusEstufas[Estufa].fimSecagem), LEN:= 2, POS:=9);
gvl_p.arrStatusEstufas[Estufa].anoSec := MID(STR:= DT_TO_STRING(gvl_p.arrStatusEstufas[Estufa].fimSecagem), LEN:= 2, POS:=6);
gvl_p.arrStatusEstufas[Estufa].horaSec := MID(STR:= DT_TO_STRING(gvl_p.arrStatusEstufas[Estufa].fimSecagem), LEN:= 2, POS:=15);
gvl_p.arrStatusEstufas[Estufa].minutoSec := MID(STR:= DT_TO_STRING(gvl_p.arrStatusEstufas[Estufa].fimSecagem), LEN:= 2, POS:=18);

///// IMPRIMIR A HORA E A DATA DO FIM DA SECAGEM --------------------------------------------------------------------------------------------------------
gvl_p.arrStatusEstufas[Estufa].statusFimSecagem := '';
gvl_p.arrStatusEstufas[Estufa].statusFimSecagem := concat(gvl_p.arrStatusEstufas[Estufa].statusFimSecagem,gvl_p.arrStatusEstufas[0].horaSec);
gvl_p.arrStatusEstufas[Estufa].statusFimSecagem := concat(gvl_p.arrStatusEstufas[Estufa].statusFimSecagem,':');
gvl_p.arrStatusEstufas[Estufa].statusFimSecagem := concat(gvl_p.arrStatusEstufas[Estufa].statusFimSecagem,gvl_p.arrStatusEstufas[0].minutoSec);
gvl_p.arrStatusEstufas[Estufa].statusFimSecagem := concat(gvl_p.arrStatusEstufas[Estufa].statusFimSecagem,' ');
gvl_p.arrStatusEstufas[Estufa].statusFimSecagem := concat(gvl_p.arrStatusEstufas[Estufa].statusFimSecagem,gvl_p.arrStatusEstufas[0].diaSec);
gvl_p.arrStatusEstufas[Estufa].statusFimSecagem := concat(gvl_p.arrStatusEstufas[Estufa].statusFimSecagem,'/');
gvl_p.arrStatusEstufas[Estufa].statusFimSecagem := concat(gvl_p.arrStatusEstufas[Estufa].statusFimSecagem,gvl_p.arrStatusEstufas[0].mesSec);
gvl_p.arrStatusEstufas[Estufa].statusFimSecagem := concat(gvl_p.arrStatusEstufas[Estufa].statusFimSecagem,'/');
gvl_p.arrStatusEstufas[Estufa].statusFimSecagem := concat(gvl_p.arrStatusEstufas[Estufa].statusFimSecagem,gvl_p.arrStatusEstufas[0].anoSec);


///// GERADOR DE LOG -------------------------------------------------------------
envialog:= 'Inicio T1 ESTUFA 021';
gvl.logRegister21:= envialog;

gvl_p.etapa_process[2]:= 'T1';

ELSE
	IF gvl_p.arr_CustomTime_021[1,1] = 0 THEN
		status:= 45;
	END_IF
	status:= 20;
END_IF

30:
tempo:= insert('T#h',INT_TO_STRING(gvl_p.arr_CustomTime_021[1,1]),2);
IF STRING_TO_DT(gvl.progInicio[Estufa]) + STRING_TO_TIME(tempo) = systemtime_to_dt(gvl.fbGetLocalSystemTime.systemTime) THEN
	status:= 31;
	
	gvl_p.zona1setpt_021:= gvl_p.arr_CustomTime_021[0,2];
	gvl_p.zona2setpt_021:= gvl_p.arr_CustomTime_021[0,2];
	gvl.progInicio[Estufa]:= DT_TO_STRING(STRING_TO_DT(gvl.progInicio[Estufa]) + STRING_TO_TIME(tempo));
	
///// GERADOR DE LOG -------------------------------------------------------------
envialog:= 'Inicio T2 ESTUFA 021';
gvl.logRegister21:= envialog;

gvl_p.etapa_process[2]:= 'T2';
	
ELSE
	status:= 30;
END_IF

31:
tempo:= insert('T#h',INT_TO_STRING(gvl_p.arr_CustomTime_021[1,2]),2);
IF STRING_TO_DT(gvl.progInicio[Estufa]) + STRING_TO_TIME(tempo) = systemtime_to_dt(gvl.fbGetLocalSystemTime.systemTime) THEN
	status:= 32;
	
	gvl_p.zona1setpt_021:= gvl_p.arr_CustomTime_021[0,3];
	gvl_p.zona2setpt_021:= gvl_p.arr_CustomTime_021[0,3];
	gvl.progInicio[Estufa]:= DT_TO_STRING(STRING_TO_DT(gvl.progInicio[Estufa]) + STRING_TO_TIME(tempo));
	
///// GERADOR DE LOG -------------------------------------------------------------
envialog:= 'Inicio T3 ESTUFA 021';
gvl.logRegister21:= envialog;

gvl_p.etapa_process[2]:= 'T3';
	
ELSE
	IF gvl_p.arr_CustomTime_021[1,2] = 0 THEN
		status:= 45;
	END_IF
	status:= 31;
END_IF

32:
tempo:= insert('T#h',INT_TO_STRING(gvl_p.arr_CustomTime_021[1,3]),2);
IF STRING_TO_DT(gvl.progInicio[Estufa]) + STRING_TO_TIME(tempo) = systemtime_to_dt(gvl.fbGetLocalSystemTime.systemTime) THEN
	status:= 33;
	
	gvl_p.zona1setpt_021:= gvl_p.arr_CustomTime_021[0,4];
	gvl_p.zona2setpt_021:= gvl_p.arr_CustomTime_021[0,4];
	gvl.progInicio[Estufa]:= DT_TO_STRING(STRING_TO_DT(gvl.progInicio[Estufa]) + STRING_TO_TIME(tempo));
	
///// GERADOR DE LOG -------------------------------------------------------------
envialog:= 'Inicio T4 ESTUFA 021';
gvl.logRegister21:= envialog;

gvl_p.etapa_process[2]:= 'T4';
	
ELSE
	IF gvl_p.arr_CustomTime_021[1,3] = 0 THEN
		status:= 45;
	END_IF
	status:= 32;
END_IF

33:
tempo:= insert('T#h',INT_TO_STRING(gvl_p.arr_CustomTime_021[1,4]),2);
IF STRING_TO_DT(gvl.progInicio[Estufa]) + STRING_TO_TIME(tempo) = systemtime_to_dt(gvl.fbGetLocalSystemTime.systemTime) THEN
	status:= 34;
	
	gvl_p.zona1setpt_021:= gvl_p.arr_CustomTime_021[0,5];
	gvl_p.zona2setpt_021:= gvl_p.arr_CustomTime_021[0,5];
	gvl.progInicio[Estufa]:= DT_TO_STRING(STRING_TO_DT(gvl.progInicio[Estufa]) + STRING_TO_TIME(tempo));
	
///// GERADOR DE LOG -------------------------------------------------------------
envialog:= 'Inicio T5 ESTUFA 021';
gvl.logRegister21:= envialog;

gvl_p.etapa_process[2]:= 'T5';
	
ELSE
	IF gvl_p.arr_CustomTime_021[1,4] = 0 THEN
		status:= 45;
	END_IF
	status:= 33;
END_IF

34:
tempo:= insert('T#h',INT_TO_STRING(gvl_p.arr_CustomTime_021[1,5]),2);
IF STRING_TO_DT(gvl.progInicio[Estufa]) + STRING_TO_TIME(tempo) = systemtime_to_dt(gvl.fbGetLocalSystemTime.systemTime) THEN
	status:= 35;
	
	gvl_p.zona1setpt_021:= gvl_p.arr_CustomTime_021[0,6];
	gvl_p.zona2setpt_021:= gvl_p.arr_CustomTime_021[0,6];
	gvl.progInicio[Estufa]:= DT_TO_STRING(STRING_TO_DT(gvl.progInicio[Estufa]) + STRING_TO_TIME(tempo));
	
///// GERADOR DE LOG -------------------------------------------------------------
envialog:= 'Inicio T6 ESTUFA 021';
gvl.logRegister21:= envialog;

gvl_p.etapa_process[2]:= 'T6';
	
ELSE
	IF gvl_p.arr_CustomTime_021[1,5] = 0 THEN
		status:= 45;
	END_IF
	status:= 34;
END_IF

35:
tempo:= insert('T#h',INT_TO_STRING(gvl_p.arr_CustomTime_021[1,6]),2);
IF STRING_TO_DT(gvl.progInicio[Estufa]) + STRING_TO_TIME(tempo) = systemtime_to_dt(gvl.fbGetLocalSystemTime.systemTime) THEN
	status:= 36;
	
	gvl_p.zona1setpt_021:= gvl_p.arr_CustomTime_021[0,7];
	gvl_p.zona2setpt_021:= gvl_p.arr_CustomTime_021[0,7];
	gvl.progInicio[Estufa]:= DT_TO_STRING(STRING_TO_DT(gvl.progInicio[Estufa]) + STRING_TO_TIME(tempo));
	
///// GERADOR DE LOG -------------------------------------------------------------
envialog:= 'Inicio T7 ESTUFA 021';
gvl.logRegister21:= envialog;

gvl_p.etapa_process[2]:= 'T7';
	
ELSE
	IF gvl_p.arr_CustomTime_021[1,6] = 0 THEN
		status:= 45;
	END_IF
	status:= 35;
END_IF

36:
tempo:= insert('T#h',INT_TO_STRING(gvl_p.arr_CustomTime_021[1,7]),2);
IF STRING_TO_DT(gvl.progInicio[Estufa]) + STRING_TO_TIME(tempo) = systemtime_to_dt(gvl.fbGetLocalSystemTime.systemTime) THEN
	status:= 37;
	
	gvl_p.zona1setpt_021:= gvl_p.arr_CustomTime_021[0,8];
	gvl_p.zona2setpt_021:= gvl_p.arr_CustomTime_021[0,8];
	gvl.progInicio[Estufa]:= DT_TO_STRING(STRING_TO_DT(gvl.progInicio[Estufa]) + STRING_TO_TIME(tempo));
	
///// GERADOR DE LOG -------------------------------------------------------------
envialog:= 'Inicio T8 ESTUFA 021';
gvl.logRegister21:= envialog;

gvl_p.etapa_process[2]:= 'T8';
	
ELSE
	IF gvl_p.arr_CustomTime_021[1,7] = 0 THEN
		status:= 45;
	END_IF
	status:= 36;
END_IF

37:
tempo:= insert('T#h',INT_TO_STRING(gvl_p.arr_CustomTime_021[1,8]),2);
IF STRING_TO_DT(gvl.progInicio[Estufa]) + STRING_TO_TIME(tempo) = systemtime_to_dt(gvl.fbGetLocalSystemTime.systemTime) THEN
	status:= 38;
	
	gvl_p.zona1setpt_021:= gvl_p.arr_CustomTime_021[0,9];
	gvl_p.zona2setpt_021:= gvl_p.arr_CustomTime_021[0,9];
	gvl.progInicio[Estufa]:= DT_TO_STRING(STRING_TO_DT(gvl.progInicio[Estufa]) + STRING_TO_TIME(tempo));
	
///// GERADOR DE LOG -------------------------------------------------------------
envialog:= 'Inicio T9 ESTUFA 021';
gvl.logRegister21:= envialog;

gvl_p.etapa_process[2]:= 'T9';
	
ELSE
	IF gvl_p.arr_CustomTime_021[1,8] = 0 THEN
		status:= 45;
	END_IF
	status:= 37;
END_IF

38:
tempo:= insert('T#h',INT_TO_STRING(gvl_p.arr_CustomTime_021[1,9]),2);
IF STRING_TO_DT(gvl.progInicio[Estufa]) + STRING_TO_TIME(tempo) = systemtime_to_dt(gvl.fbGetLocalSystemTime.systemTime) THEN
	status:= 40;
	
	gvl_p.zona1setpt_021:= gvl_p.arr_CustomTime_021[0,10];
	gvl_p.zona2setpt_021:= gvl_p.arr_CustomTime_021[0,10];
	gvl.progInicio[Estufa]:= DT_TO_STRING(STRING_TO_DT(gvl.progInicio[Estufa]) + STRING_TO_TIME(tempo));
	
///// GERADOR DE LOG -------------------------------------------------------------
envialog:= 'Inicio T10 ESTUFA 021';
gvl.logRegister21:= envialog;

gvl_p.etapa_process[2]:= 'T10';
	
ELSE
	IF gvl_p.arr_CustomTime_021[1,9] = 0 THEN
		status:= 45;
	END_IF
	status:= 38;
END_IF

40:
tempo:= insert('T#h',INT_TO_STRING(gvl_p.arr_CustomTime_021[1,10]),2);
IF STRING_TO_DT(gvl.progInicio[Estufa]) + STRING_TO_TIME(tempo) = systemtime_to_dt(gvl.fbGetLocalSystemTime.systemTime) THEN
	status:= 50;
	
	gvl_p.arrStatusEstufas[Estufa].startManual:= FALSE;
	gvl.bstartchart021:= FALSE;
	gvl.desl_aquecimento_021:= TRUE;
	fbTimeAqueci(in:=TRUE, pt:=T#1S);
	
	gvl_p.etapa_process[Estufa] := '';
	
	gvl_p.arrStatusEstufas[Estufa].statusInicioSecagem := '';
	gvl_p.arrStatusEstufas[Estufa].inicioReator := '';
	gvl_p.arrStatusEstufas[Estufa].statusFimSecagem := '';
	gvl_p.arrStatusEstufas[Estufa].statusFimArmazenagem := '';
	gvl_p.arrStatusEstufas[Estufa].fimSecagem:= DT#1970-1-1-0:0:0;
	gvl.endArm21:= T#0S;
	gvl.endSeca21:= T#0S;
	
///// GERADOR DE LOG -------------------------------------------------------------
envialog:= 'Programação Finalizada ESTUFA 021';
gvl.logRegister21:= envialog;

gvl_p.etapa_process[2]:= '';

ELSE
	IF gvl_p.arr_CustomTime_021[1,10] = 0 THEN
		status:= 45;
	END_IF
	status:= 40;
END_IF

45:
IF gvl_p.arrStatusEstufas[Estufa].startManual THEN
status:= 50;
	
	gvl_p.arrStatusEstufas[Estufa].startManual:= FALSE;
	gvl.bstartchart021:= FALSE;
	gvl.desl_aquecimento_021:= TRUE;
	fbTimeAqueci(in:=TRUE, pt:=T#1S);
	
	gvl_p.etapa_process[Estufa] := '';
	
	gvl_p.arrStatusEstufas[Estufa].statusInicioSecagem := '';
	gvl_p.arrStatusEstufas[Estufa].inicioReator := '';
	gvl_p.arrStatusEstufas[Estufa].statusFimSecagem := '';
	gvl_p.arrStatusEstufas[Estufa].statusFimArmazenagem := '';
	gvl_p.arrStatusEstufas[Estufa].fimSecagem:= DT#1970-1-1-0:0:0;
	gvl.endArm21:= T#0S;
	gvl.endSeca21:= T#0S;
	
///// GERADOR DE LOG -------------------------------------------------------------
envialog:= 'Programação Finalizada ESTUFA 021';
gvl.logRegister21:= envialog;

gvl_p.etapa_process[2]:= '';

ELSE
	status:= 45;
END_IF

50:
IF fbTimeAqueci.Q THEN
	status:= 0;
	
	gvl.desl_aquecimento_021:= FALSE;
	fbTimeAqueci(in:= FALSE);
	
ELSE
	status:= 50;
END_IF
END_CASE

END_PROGRAM

// ---- POUs/POU_Persistent.TcPOU
PROGRAM POU_Persistent
VAR
	fbWritePersistentData: FB_WritePersistentData;
	bPersistentWr: BOOL;
	
END_VAR


fbWritePersistentData(
	NETID:= , 
	PORT:= 851 , 
	START:= bPersistentWr, 
	TMOUT:= , 
	MODE:= , 
	BUSY=> , 
	ERR=> , 
	ERRID=> );
	
bPersistentWr:= FALSE;

END_PROGRAM

// ---- POUs/P_TextModeWrite.TcPOU
(* Writing of CSV file in text mode. None of the field value is containing any non-printing control characters like line feed, carriage return, quotation marks, semicolon... *)
PROGRAM P_TextModeWrite
VAR_INPUT
	
	bWrite			: BOOL := FALSE;(* Rising edge starts program execution *)
	sNetId			: T_AmsNetId := '';	(* TwinCAT system network address *)
	sFileName		: T_MaxString := '\Hard Disk\ftp\GloboReport.csv';(* CSV destination file path and name *)
	sCSVLine		: T_MaxString := '';(* Single CSV text line (row, record), we are using string as record buffer (your are able to see created fields) *)
	sCSVField		: T_MaxString := '';(* Single CSV field value (column, record field) *)
	bBusy			: BOOL;
	bError			: BOOL;
	nErrId			: UDINT;
	nRow	 		: UDINT 	:= 0;(* Row number (record) *)
	nColumn			: UDINT 	:= 0;(* Column number (record field) *)
	hFile			: UINT		:= 0;(* File handle of the source file *)
	step			: DWORD 	:= 0;
	fbFileOpen		: FB_FileOpen;(* Opens file *)
	fbFileClose		: FB_FileClose;(* Closes file *)
	fbFilePuts		: FB_FilePuts;(* Writes one record (line) *)
	fbWriter		: FB_CSVMemBufferWriter;(* Helper function block used to create CSV data bytes (single record line) *)

	database		: ARRAY[0..MAX_CSV_ROWS, 0..MAX_CSV_COLUMNS ] OF STRING(MAX_CSV_FIELD_LENGTH);  (* Source PLC database *)
	(*'0_0', '0_1', '0_2', '0_3', '0_4', '0_5',
	'1_0', '1_1', '1_2', '1_3', '1_4', '1_5',
	'2_0', '2_1', '2_2', '2_3', '2_4', '2_5',
	'3_0', '3_1', '3_2', '3_3', '3_4', '3_5',
	'4_0', '4_1', '4_2', '4_3', '4_4', '4_5',
	'5_0', '5_1', '5_2', '5_3', '5_4', '5_5'];*)

END_VAR

CASE step OF
	0:	(* Wait for rising edge at bWrite variable *)
		IF bWrite THEN
			bWrite 	:= FALSE;
			bBusy 	:= TRUE;
			bError	:= FALSE;
			nErrId	:= 0;
			hFile	:= 0;
			nRow	:= 0;
			nColumn	:= 0;
			step 	:= 1;
			ReportGenerator();
		END_IF

	1:	(* Open source file *)
		fbFileOpen(  bExecute := FALSE  );
		fbFileOpen( sNetId := sNetId, sPathName := sFileName, nMode := FOPEN_MODEWRITE OR FOPEN_MODETEXT,(* Open file in TEXT mode! *)
					ePath := PATH_GENERIC, bExecute := TRUE );
		step := 2;

	2:(* Wait until open not busy *)
		fbFileOpen( bExecute := FALSE, bError => bError, nErrID => nErrID, hFile => hFile );
		IF NOT fbFileOpen.bBusy THEN
			IF NOT fbFileOpen.bError THEN
				step := 3;
			ELSE(* Error: file not found? *)
				step := 100;
			END_IF
		END_IF

	3:(* Convert one PLC record to CSV format *)
		sCSVLine := '';
		fbWriter.eCmd := eEnumCmd_First;(* Write first field value *)
		IF nRow <= main.nRecords THEN
		
	
			FOR nColumn := 0 TO MAX_CSV_COLUMNS BY 1 DO

				sCSVField := STRING_TO_CSVFIELD( gvl.database[ nRow, nColumn ], FALSE );(* TODO: Get field value from your application *)

				(* Add new field to the record buffer *)
				fbWriter( 	pBuffer := ADR( sCSVLine ), cbBuffer := SIZEOF( sCSVLine ) - 1, putValue := sCSVField, pValue := 0, cbValue := 0,
							bCRLF := ( nColumn = MAX_CSV_COLUMNS ) );(* bCRLF == TRUE => Write CRLF after the last field value *)
				IF fbWriter.bOk THEN
					fbWriter.eCmd := eEnumCmd_Next;(* Write next field value *)
				ELSE(* Error *)
					step := 100;
					RETURN;
				END_IF

			END_FOR(* FOR nColumn := 0... *)

			(* FB_FilePuts adds allready CR (carriage return) to the written line.
			We have to replace the $R$L characters with $L character to avoid double CR. *)
			IF RIGHT( sCSVLine, 2 ) = '$R$L' THEN
				sCSVLine := REPLACE( sCSVLine, '$L', 2, LEN( sCSVLine ) - 1 );
			END_IF

			nRow := nRow + 1;(* Increment number of created records (rows) *)
			step := 4;(* Write record to the file *)
		
		ELSE(* All rows written => Close file *)
			step := 10;
		END_IF

	4:	(* Write single text line *)
		fbFilePuts( bExecute := FALSE );
		fbFilePuts( sNetId := sNetId, hFile := hFile, sLine := sCSVLine, bExecute := TRUE );
		step := 5;

	5:(* Wait until write not busy *)
		fbFilePuts( bExecute := FALSE, bError => bError, nErrID => nErrID );
		IF NOT fbFilePuts.bBusy THEN
			IF NOT fbFilePuts.bError THEN
				step := 3;(* Write next record *)
			ELSE(* Error *)
				step := 100;
			END_IF
		END_IF

	10:	(* Close source file *)
		fbFileClose( bExecute := FALSE );
		fbFileClose( sNetId := sNetId, hFile := hFile, bExecute := TRUE );
		step := 11;

	11:(* Wait until close not busy *)
		fbFileClose( bExecute := FALSE, bError => bError, nErrID => nErrID );
		IF ( NOT fbFileClose.bBusy ) THEN
			hFile := 0;
			step := 100;
		END_IF

	100: (* Error or ready step => cleanup *)
		IF ( hFile <> 0 ) THEN
			step := 10; (* Close the source file *)
		ELSE
			bBusy := FALSE;
			step := 0;	(* Ready *)
		END_IF

END_CASE

END_PROGRAM

// ---- POUs/ReportGenerator.TcPOU
PROGRAM ReportGenerator
VAR
	i: UDINT;
	letraD: INT;
	letraH: INT;
	letraM: INT;
	
END_VAR


gvl.database[0,0]:= 'Data';
gvl.database[0,1]:= 'Hora';
gvl.database[0,2]:= 'Ordem Fabri';
gvl.database[0,3]:= 'Lote';
gvl.database[0,4]:= 'Posicao';
gvl.database[0,5]:= 'Reator';
gvl.database[0,6]:= 'Tempo em Processo';
gvl.database[0,7]:= 'Temperatura';
gvl.database[0,8]:= 'Automatico';
gvl.database[0,9]:=	'Classe';
gvl.database[0,10]:='Fat. Potencia';
gvl.database[0,11]:='Isolamento';
gvl.database[0,12]:='Potencia';


FOR i:=1 TO MAX_CSV_ROWS BY 1 DO
gvl.database[i,0]:= gvl.aSelect19[i].data;
gvl.database[i,1]:= gvl.aSelect19[i].hora;
gvl.database[i,2]:= gvl.aSelect19[i].orfb;
gvl.database[i,3]:= gvl.aSelect19[i].lote;
gvl.database[i,4]:= gvl.aSelect19[i].pos;
gvl.database[i,5]:= gvl.aSelect19[i].reator;
gvl.aSelect19[i].tempo:= delete(gvl.aSelect19[i].tempo,2,1);
gvl.database[i,6]:= gvl.aSelect19[i].tempo;
gvl.database[i,7]:= LREAL_TO_STRING(gvl.aSelect19[i].temp);
gvl.database[i,8]:= gvl.aSelect19[i].auto;
gvl.database[i,9]:= gvl.aSelect19[i].class;
gvl.database[i,10]:= gvl.aSelect19[i].fPot;
gvl.database[i,11]:= LREAL_TO_STRING(gvl.aSelect19[i].isola);
gvl.database[i,12]:= INT_TO_STRING(REAL_TO_INT(gvl.aSelect19[i].pot));
END_FOR

END_PROGRAM

// ---- GlobalTextList.TcGTLO
TEXTLIST GlobalTextList
  820 = '        203/020'
  674 = '        203/021'
  492 = '       203/019'
  604 = '       203/020'
  1072 = '       203/021'
  536 = '     203/019'
  643 = '%'
  213 = '%.'
  249 = '%.01f'
  115 = '%.1'
  939 = '%.1f'
  567 = '%.2f'
  805 = '%1f'
  825 = '%1f.'
  746 = '%d'
  1002 = '%d º'
  546 = '%dt'
  1289 = '%f'
  50 = '%i'
  969 = '%i º'
  89 = '%r º'
  400 = '%s'
  116 = '%s Etapa do processo'
  51 = '%t'
  289 = '%t[d MMM yy HH:mm]'
  1177 = '%t[]'
  694 = '%[d MMM yy HH:mm]'
  998 = '-'
  960 = '019'
  929 = '020'
  729 = '021'
  787 = '10'
  744 = '12'
  916 = '120'
  823 = '120º'
  211 = '12345'
  423 = '13:00:30 20/02/2024'
  541 = '18'
  617 = '2024'
  1015 = '203'
  731 = '203/019'
  419 = '203/020'
  240 = '203/021'
  470 = '31'
  430 = '40'
  1007 = ':'
  245 = 'Adicionar'
  1475 = 'Adicionar comentário ao Log'
  1014 = 'Adicionar Reator'
  798 = 'Admin'
  899 = 'Agendar Início?'
  876 = 'Ajustar Data de Início do Programa'
  250 = 'Alarme'
  863 = 'Ano'
  700 = 'Aquecimento'
  11 = 'Aquecimento Desligado'
  995 = 'Aquecimento Ligado'
  554 = 'Armazenagem:'
  1310 = 'ATENÇÃO!\nA adição de reatores agora irá alterar o término da programação ativa. Confirma a adição de um reator na posição     do carrinho?'
  133 = 'ATENÇÃO!\nA adição de reatores agora irá alterar o término da programação ativa. Deseja continuar com a adição de um reator?'
  444 = 'ATENÇÃO!\nA adição de um reator agora irá alterar o término da programação ativa. Deseja continuar com a adição de um reator?'
  650 = 'ATENÇÃO!Confirma a adição de um reator na posição     do carrinho?'
  834 = 'Cancela'
  451 = 'Cancelar'
  919 = 'Carregamento'
  113 = 'celsios'
  994 = 'Classe'
  1173 = 'Classe de Isolamento:'
  388 = 'Classe de Tensão:'
  246 = 'Classe:'
  575 = 'Configuração %s'
  330 = 'Configuração Posição'
  440 = 'Configuração Posição 01'
  1440 = 'Confirma'
  96 = 'Confirma a adição de um reator na posição     do carrinho?'
  313 = 'Confirma a finalização da programação?'
  959 = 'Confirma o inicio de um programa com:'
  1385 = 'Confirmar o início do programa para a Estufa %s com as seguintes configurações?'
  688 = 'Confirmar o início do programa para a Estufa 203/019 com as seguintes configurações?'
  571 = 'Continuar'
  416 = 'Dashboard'
  532 = 'Data'
  1391 = 'Data:'
  760 = 'Defina a temperatura e o tempo que ela ficará ativa. '
  1044 = 'Desliga Ciclo de Aquecimento'
  171 = 'Dia'
  609 = 'Edite a data de inicio do programa:'
  150 = 'Edite o tempo de secagem'
  681 = 'Edite o tempo de secagem:'
  772 = 'Estufa 01'
  260 = 'Estufa 02'
  539 = 'Estufa 203/019'
  502 = 'Estufa 203/020'
  1056 = 'Estufa 203/021'
  1685 = 'Estufa:'
  531 = 'Eventos'
  144 = 'ewfqreg'
  713 = 'Falha Temperatura Alta'
  696 = 'Filtro:'
  733 = 'Fim da Armasenagem:'
  804 = 'Fim da Armazenagem:'
  716 = 'Fim da Secagem:'
  786 = 'Fim de Ciclo de Aquecimento'
  117 = 'Fim de Ciclo de AquecimentoDesligado'
  511 = 'final'
  383 = 'Finaliza Programação'
  776 = 'FP:'
  176 = 'Gerador de Histórico'
  1932 = 'Gerando'
  441 = 'Gerando ...'
  970 = 'Gerar Histórico'
  693 = 'Graus'
  429 = 'Grava Posição'
  603 = 'Gravar Posição'
  648 = 'Gráfico'
  891 = 'Gráfico de Acompanhamento da Temperatura'
  726 = 'Gráficos'
  2010 = 'GVL.arrCVSfilter[GVL.radioEstufa].dia'
  515 = 'Histórico'
  1057 = 'Hora:'
  41 = 'Horas'
  544 = 'Horas:'
  367 = 'Iniciar'
  422 = 'Inícia Programação'
  652 = 'Início da Secagem:'
  230 = 'Início de Programa'
  1058 = 'Início:'
  752 = 'Legenda'
  1348 = 'Letra'
  220 = 'Liga Ciclo de Aquecimento'
  453 = 'Liga Ventilação'
  684 = 'Limpar Gráfico'
  545 = 'Limpar Posição'
  817 = 'Limpar Tela'
  848 = 'LogIn'
  1313 = 'LogOut'
  1164 = 'Lote'
  1507 = 'Lote:'
  1033 = 'Manutenção'
  1618 = 'Mês'
  917 = 'None'
  450 = 'Numero'
  15 = 'Numero de Série:'
  521 = 'Numero OF:'
  655 = 'NÃO'
  736 = 'Número'
  476 = 'OF'
  705 = 'Operator'
  1068 = 'Ordem de Fabricação'
  940 = 'Posição de Reator Ocupada'
  378 = 'Posição Livre'
  484 = 'Posição Ocupada Com Reator'
  678 = 'Posição Ocupada COM Reator'
  958 = 'Posição ocupada por completo'
  806 = 'Posição Ocupada Sem Reator'
  290 = 'Posição Ocupada SEM Reator'
  288 = 'Possui Reator'
  685 = 'Potência:'
  498 = 'Programação'
  962 = 'Programação Estufa 203/019'
  1514 = 'Programação Manual'
  493 = 'Purgando Câmara'
  526 = 'Qtd. Pos. Utilizadas:'
  941 = 'Queimador 1 Bloqueado'
  928 = 'Queimador 2 Bloqueado'
  895 = 'Reator'
  857 = 'Secagem'
  1242 = 'Secagem Reator'
  119 = 'Secagem:'
  28 = 'Segurança'
  673 = 'Service'
  630 = 'Set Point'
  725 = 'Set Point:'
  236 = 'SIM'
  387 = 'Sistema Supervisório de Estufas'
  125 = 'Sobrecarga Motor 1 de Ventilação'
  829 = 'Sobrecarga Motor 2 de Ventilação'
  662 = 'Sobrecarga Motor do Exaustor de Purga'
  362 = 'Status da Programação'
  988 = 'Status de cada posição'
  103 = 'Série:'
  734 = 'tab'
  479 = 'TabTest'
  1254 = 'TEMPERATURA'
  1426 = 'TEMPERATURA (ºC)'
  229 = 'Temperatura Atual:'
  983 = 'Temperatura de Armazenagem:'
  449 = 'Temperatura de Secagem:'
  735 = 'Temperatura de Segurança'
  225 = 'Temperatura Segurança'
  542 = 'Temperatura Zona 1'
  170 = 'Temperatura Zona 1:'
  296 = 'Temperatura Zona 2'
  560 = 'Temperatura Zona 2:'
  343 = 'TEMPERATURA ºC'
  759 = 'TemperaturSegurança'
  1699 = 'TEMPO'
  1036 = 'TEMPO (H)'
  931 = 'Tempo de Armazenagem:'
  822 = 'Tempo de Secagem:'
  12 = 'Tempo Restante'
  434 = 'Tempo Restante:'
  1025 = 'Tempo total:'
  1375 = 'Tensão Nominal:'
  534 = 'Test2'
  778 = 'Total de posições:'
  283 = 'Total de Posições:'
  585 = 'Total de Reatores:'
  443 = 'Unidades'
  915 = 'Ventilação'
  918 = 'Ventilação Ligada'
  40 = 'xfdsfg'
  414 = 'ºC'
END_TEXTLIST

// ---- VISUs/Aba_Estufa.TcVIS
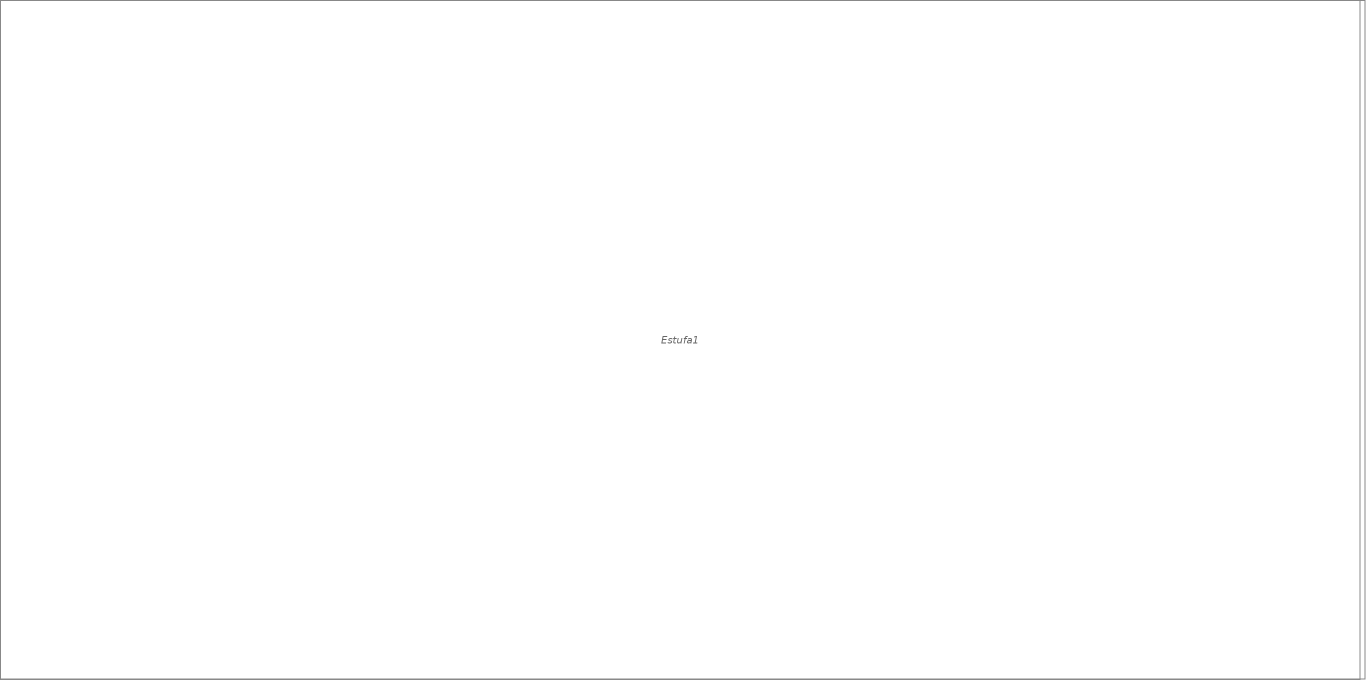
VISUALIZATION Aba_Estufa  // 1366x680
    TabControl (0,0 1360x680)
        shows Estufa1()
        shows Grafico()
        [0]: TabTitle=Dashboard
        [1]: TabTitle=Gráfico
END_VISUALIZATION

// ---- VISUs/Aba_Estufa_2.TcVIS
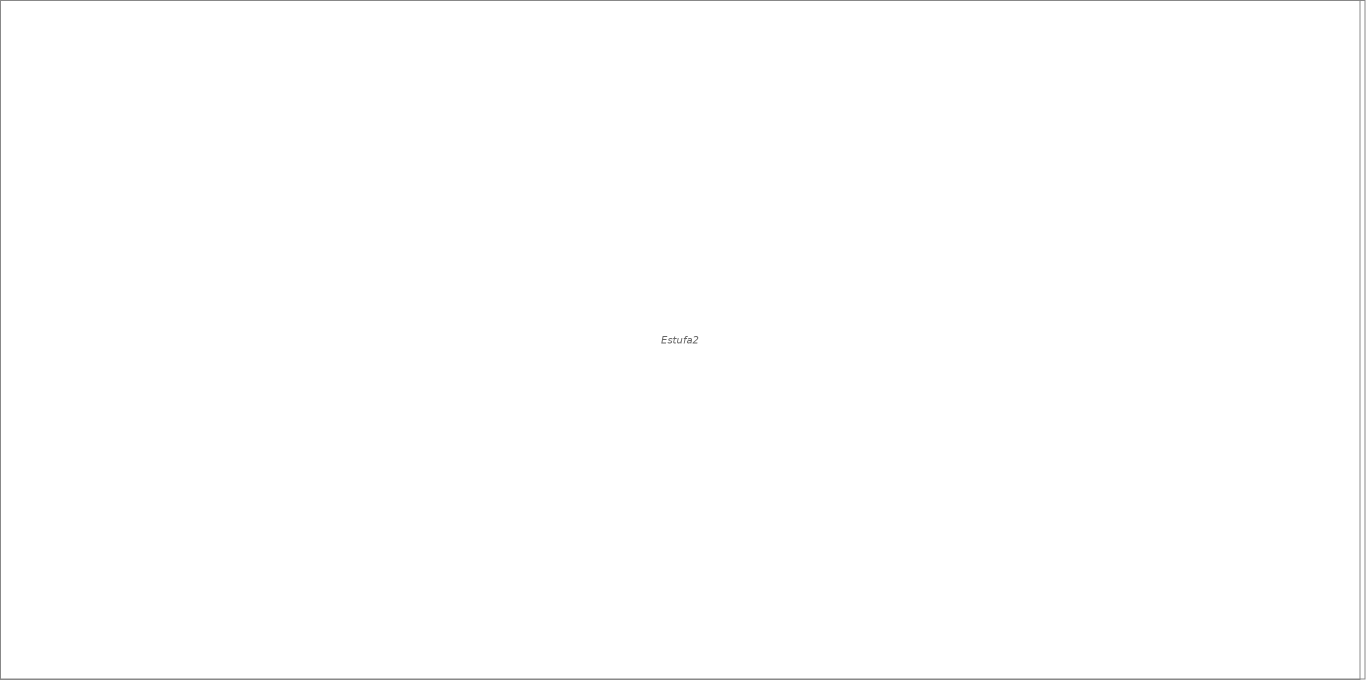
VISUALIZATION Aba_Estufa_2  // 1366x680
    TabControl (0,0 1360x680)
        shows Estufa2()
        shows Grafico_2()
        [0]: TabTitle=Dashboard
        [1]: TabTitle=Gráfico
END_VISUALIZATION

// ---- VISUs/Aba_Manu.TcVIS
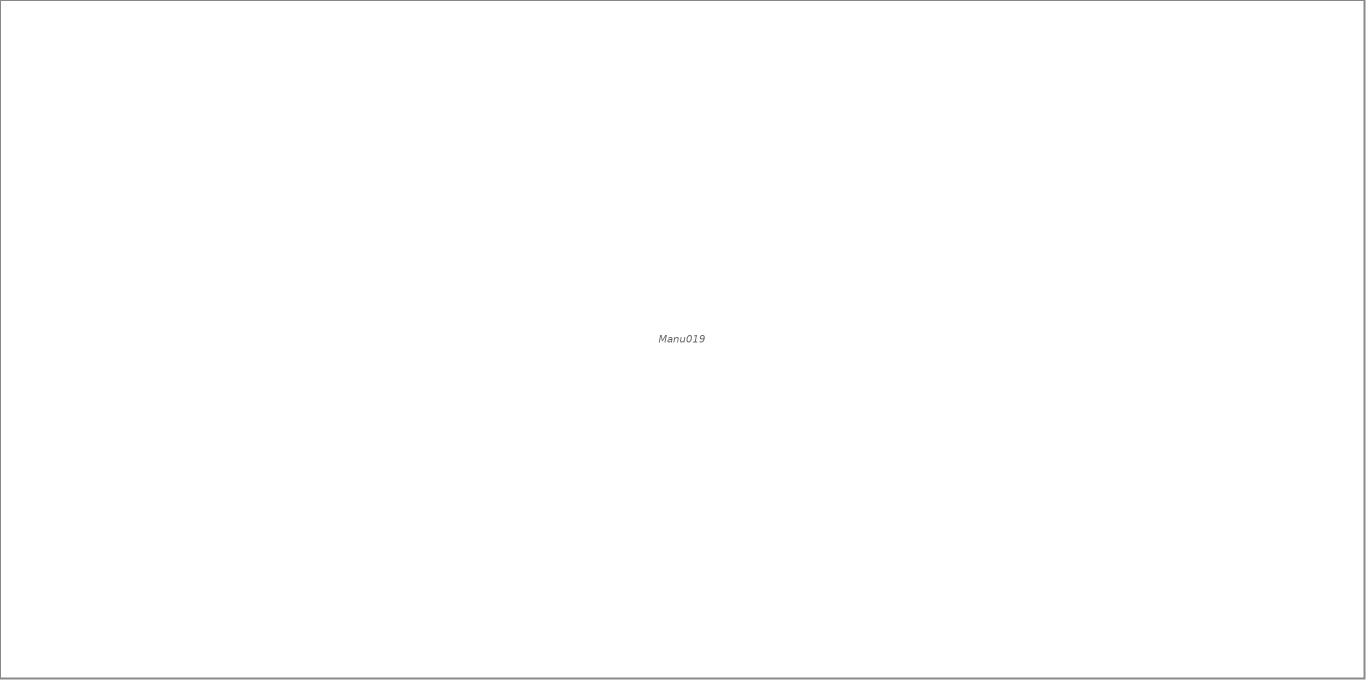
VISUALIZATION Aba_Manu  // 1366x680
    TabControl (0,0 1364x678)
        shows Manu019()
        shows Manu020()
        shows Manu021()
        [0]: TabTitle=203/019
        [1]: TabTitle=203/020
        [2]: TabTitle=203/021
END_VISUALIZATION

// ---- VISUs/addComment.TcVIS
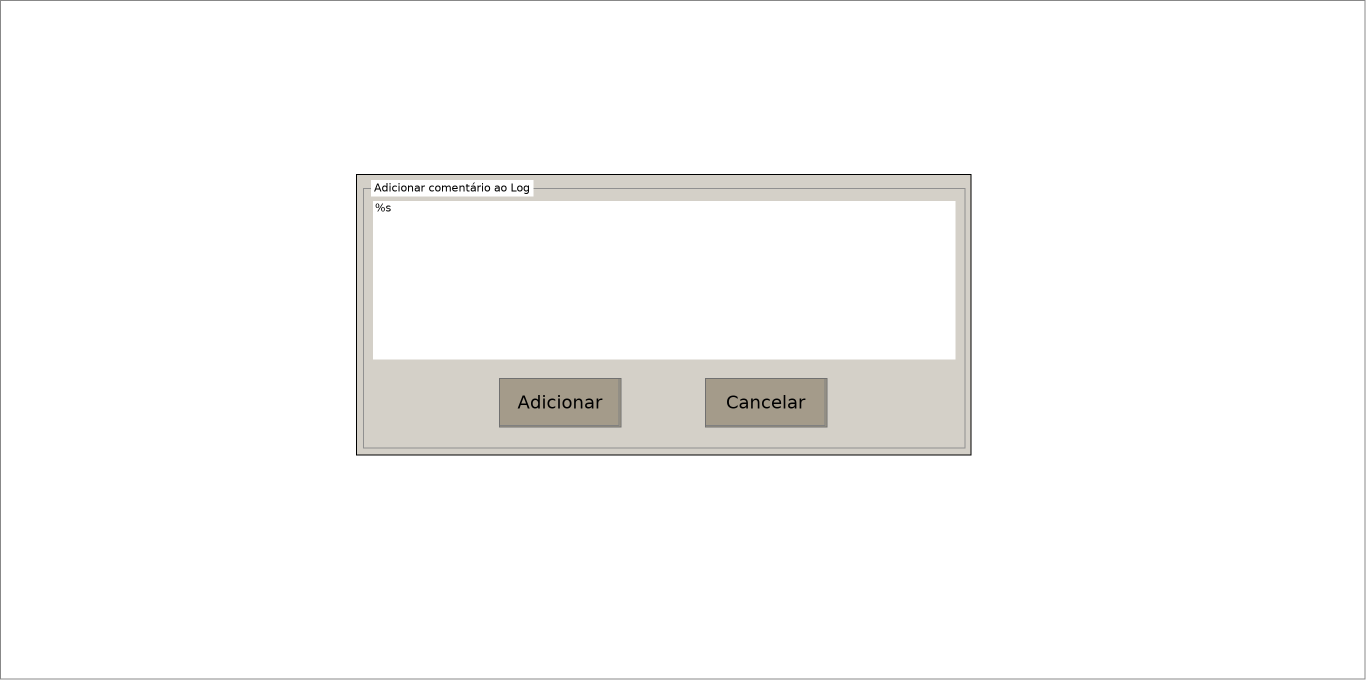
VISUALIZATION addComment  // 1366x680
    Rectangle (356,174 615x281)
    GroupBox (363,180 602x268), "Adicionar comentário ao Log"
        Textfield (9,20 584x160), "%s", text variable: GVL.addTextLog
            OnMouseDown: write GVL.addTextLog via VisuDialogs.Keypad, format ADD COMMENT
        Button (136,198 122x49), "Adicionar"
            OnMouseClick: CloseDialog Dialog=addComment, Result=OK, NumpadKeypadSet=True
            OnMouseClick: execute {
                ///// GERADOR DE LOG -------------------------------------------------------------
                IF GVL.actEst = 0 THEN
                	gvl.logRegister19:= gvl.addTextLog;
                END_IF
                IF GVL.actEst = 1 THEN
                	gvl.logRegister20:= gvl.addTextLog;
                END_IF
                IF GVL.actEst = 2 THEN
                	gvl.logRegister21:= gvl.addTextLog;
                END_IF
            }
        Button (342,198 122x49), "Cancelar"
            OnMouseClick: CloseDialog Dialog=addComment, Result=OK, NumpadKeypadSet=True
END_VISUALIZATION

// ---- VISUs/ConfigPosicao_3.TcVIS
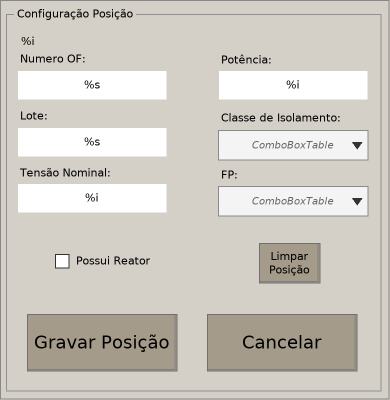
VISUALIZATION ConfigPosicao_3  // 390x400
VAR_IN_OUT
	bReator: BOOL;
	iOFnumber: INT;
	iSrlNumber: INT;
	
	
	
END_VAR
    GroupBox (6,6 375x385), "Configuração Posição"
        Checkbox (47,242 110x26), "Possui Reator", variable: gravarConfigPosicao021.bReator[2]
        Label (11,38 81x30), "Numero OF:"
        Textfield (11,64 150x30), "%s", text variable: GVL.cfgPos_OF021
            OnMouseDown: write the text variable via VisuDialogs.Numpad
        Label (11,152 103x30), "Tensão Nominal:"
        Button (21,308 150x57), "Gravar Posição"
            OnMouseClick: CloseDialog Dialog=ConfigPosicao_3, Result=OK, NumpadKeypadSet=True
            OnMouseClick: execute { gravarConfigPosicao021(); }
        Button (201,308 150x57), "Cancelar"
            OnMouseClick: CloseDialog Dialog=ConfigPosicao_3, Result=Cancel, NumpadKeypadSet=True
        Button (253,237 61x40), "Limpar Posição"
            OnMouseClick: CloseDialog Dialog=ConfigPosicao_3, Result=Cancel, NumpadKeypadSet=True
            OnMouseClick: execute {
                IF gvl_p.aPositionsE021[gvl.actPos].cor = 1
                OR gvl_p.aPositionsE021[gvl.actPos].cor = 2 THEN
                IF gvl.totalPos[2] > 0 THEN
                gvl.totalPos[2]:= gvl.totalPos[2]-1;
                END_IF
                END_IF
                gvl_p.aPositionsE021[gvl.actPos].numOF:='0';
                gvl_p.aPositionsE021[gvl.actPos].lote:='0';
                gvl_p.aPositionsE021[gvl.actPos].class:=0;
                gvl_p.aPositionsE021[gvl.actPos].pot:=0;
                gvl_p.aPositionsE021[gvl.actPos].cor:=0;
                gvl_p.aPositionsE021[gvl.actPos].text:='';
                bReator:=false;
                ///// GERADOR DE LOG -------------------------------------------------------------
                gvl.envialog:= 'Posição Nº ';
                gvl.envialog:= concat(gvl.envialog, INT_TO_STRING(gvl.actPos));
                gvl.envialog:= concat(gvl.envialog,' foi limpa. ESTUFA 021');
                gvl.logRegister21:= gvl.envialog;
            }
        Textfield (212,64 150x30), "%i", text variable: GVL.cfgPos_Pot021
            OnMouseDown: write the text variable via VisuDialogs.Numpad
        Label (11,95 81x30), "Lote:"
        Label (212,154 56x30), "FP:"
        Label (212,97 144x30), "Classe de Isolamento:"
        Textfield (11,177 150x30), "%i", text variable: GVL.cfgPos_Class021
            OnMouseDown: write the text variable via VisuDialogs.Numpad
    Label (218,45 56x30), "Potência:"
    Rectangle (17,30 22x23), "%i", text variable: GVL.actPos
    Textfield (17,127 150x30), "%s", text variable: GVL.cfgPos_LT021
        OnMouseDown: write the text variable via VisuDialogs.Keypad
    ComboBoxTable (218,130 150x30), variable: GVL.cfgPos_Iso021, data array: GVL_P.arr_Iso_3
        p3854506369: GVL_P.arr_Iso_3[INDEX]
    ComboBoxTable (218,186 150x30), variable: GVL.cfgPos_FP021, data array: GVL_P.arr_FP_3
        p3854506369: GVL_P.arr_FP_3[INDEX]
END_VISUALIZATION

// ---- VISUs/ConfigPosicao_2.TcVIS
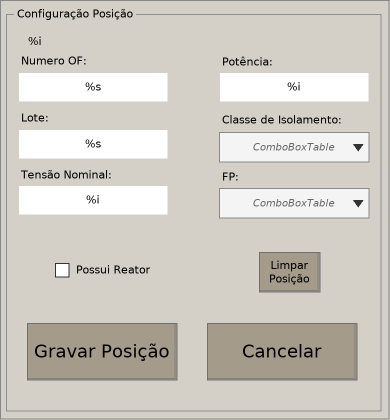
VISUALIZATION ConfigPosicao_2  // 390x420
VAR_IN_OUT
	bReator: BOOL;
	iOFnumber: INT;
	iSrlNumber: INT;
	
	
	
END_VAR
    GroupBox (6,6 375x405), "Configuração Posição"
        Checkbox (47,251 110x26), "Possui Reator", variable: gravarConfigPosicao020.bReator[1]
        Button (21,317 150x57), "Gravar Posição"
            OnMouseClick: CloseDialog Dialog=ConfigPosicao_2, Result=OK, NumpadKeypadSet=True
            OnMouseClick: execute { gravarConfigPosicao020(); }
        Button (201,317 150x57), "Cancelar"
            OnMouseClick: CloseDialog Dialog=ConfigPosicao_2, Result=Cancel, NumpadKeypadSet=True
        Button (253,246 61x40), "Limpar Posição"
            OnMouseClick: CloseDialog Dialog=ConfigPosicao_2, Result=Cancel, NumpadKeypadSet=True
            OnMouseClick: execute {
                gvl_p.aPositionsE020[gvl.actPos].numOF:='0';
                gvl_p.aPositionsE020[gvl.actPos].lote:='0';
                gvl_p.aPositionsE020[gvl.actPos].class:=0;
                gvl_p.aPositionsE020[gvl.actPos].pot:=0;
                gvl_p.aPositionsE020[gvl.actPos].cor:=0;
                IF gvl.totalPos[gvl.actEst] <> 0 THEN
                gvl.totalPos[gvl.actEst]:= gvl.totalPos[gvl.actEst] - 1;
                ELSE
                	gvl.totalPos[gvl.actEst] := 0;
                END_IF
                bReator:=false;
                ///// GERADOR DE LOG -------------------------------------------------------------
                gvl.envialog:= 'Posição Nº ';
                gvl.envialog:= concat(gvl.envialog, INT_TO_STRING(gvl.actPos));
                gvl.envialog:= concat(gvl.envialog,' foi limpa. ESTUFA 020');
                gvl.logRegister20:= gvl.envialog;
            }
        Label (12,40 81x30), "Numero OF:"
    Rectangle (24,30 22x23), "%i", text variable: GVL.actPos
    Textfield (18,72 150x30), "%s", text variable: GVL.cfgPos_OF020
        OnMouseDown: write the text variable via VisuDialogs.Numpad
    Label (18,160 104x30), "Tensão Nominal:"
    Textfield (219,72 150x30), "%i", text variable: GVL.cfgPos_Pot020
        OnMouseDown: write the text variable via VisuDialogs.Numpad
    Label (18,103 81x30), "Lote:"
    Label (219,162 56x30), "FP:"
    Label (219,105 144x30), "Classe de Isolamento:"
    Textfield (18,185 150x30), "%i", text variable: GVL.cfgPos_Class020
        OnMouseDown: write the text variable via VisuDialogs.Numpad
    Label (219,47 56x30), "Potência:"
    Textfield (18,129 150x30), "%s", text variable: GVL.cfgPos_LT020
        OnMouseDown: write the text variable via VisuDialogs.Keypad
    ComboBoxTable (219,132 150x30), variable: GVL.cfgPos_Iso020, data array: GVL_P.arr_Iso_2
        p3854506369: GVL_P.arr_Iso_2[INDEX]
    ComboBoxTable (219,188 150x30), variable: GVL.cfgPos_FP020, data array: GVL_P.arr_FP_2
        p3854506369: GVL_P.arr_FP_2[INDEX]
END_VISUALIZATION

// ---- VISUs/ConfigPosicao_Reator.TcVIS
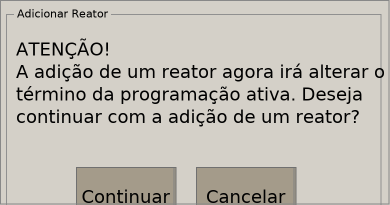
VISUALIZATION ConfigPosicao_Reator  // 390x205
VAR_IN_OUT
	bReator: BOOL;
	iOFnumber: INT;
	iSrlNumber: INT;
	
	
	
END_VAR
    GroupBox (6,6 375x193), "Adicionar Reator"
        Label (22,31 332x63), "Confirma a adição de um reator na posição do carrinho?"
        Button (21,106 95x60), "Gravar Posição"
            OnMouseClick: CloseDialog Dialog=ConfigPosicao_Reator, Result=OK, NumpadKeypadSet=True
            OnMouseClick: execute { gravarConfigPosicao_Reator(); }
        Button (141,106 95x60), "Cancelar"
            OnMouseClick: CloseDialog Dialog=ConfigPosicao_Reator, Result=Cancel, NumpadKeypadSet=True
        Rectangle (96,54 22x23), "%i", text variable: GVL.actReat
        Button (261,106 95x60), "Limpar Posição"
            OnMouseClick: CloseDialog Dialog=ConfigPosicao, Result=Cancel, NumpadKeypadSet=True
            OnMouseClick: execute { gvl_p.corPosReator1[gvl.actReat].cor:= 0; }
    Frame (0,0 390x255), invisible if: posCarrinho.bNotificaTime
        shows Notifica24horas()
END_VISUALIZATION

// ---- VISUs/ConfigPosicao_Reator_2.TcVIS
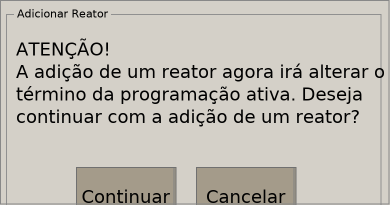
VISUALIZATION ConfigPosicao_Reator_2  // 390x205
VAR_IN_OUT
	bReator: BOOL;
	iOFnumber: INT;
	iSrlNumber: INT;
	
	
	
END_VAR
    GroupBox (6,6 375x193), "Adicionar Reator"
        Label (22,31 332x63), "Confirma a adição de um reator na posição do carrinho?"
        Button (21,106 95x60), "Gravar Posição"
            OnMouseClick: CloseDialog Dialog=ConfigPosicao_Reator_2, Result=OK, NumpadKeypadSet=True
            OnMouseClick: execute { gravarConfigPosicao_Reator_2(); }
        Button (141,106 95x60), "Cancelar"
            OnMouseClick: CloseDialog Dialog=ConfigPosicao_Reator_2, Result=Cancel, NumpadKeypadSet=True
        Rectangle (96,54 22x23), "%i", text variable: GVL.actReat
        Button (261,106 95x60), "Limpar Posição"
            OnMouseClick: CloseDialog Dialog=ConfigPosicao_Reator_2, Result=Cancel, NumpadKeypadSet=True
            OnMouseClick: execute { gvl_p.corPosReator2[gvl.actReat].cor:= 0; }
    Frame (0,0 390x255), invisible if: posCarrinho2.bNotificaTime
        shows Notifica24horas()
END_VISUALIZATION

